		ExchangeData(	ADR(Parameters.Regulation.ExtractAir.ControlMode), 
						ADR(ADS_Standard.Tags.Settings.ExtractFanControlMode), 
						SIZEOF(Parameters.Regulation.ExtractAir.ControlMode), 
						ADR(SavedParameters.Regulation.Temperature.TemperatureControlSource), 
						ADR(SavedInterface.ExtractFanControlMode), 
						'INT', ('Parameters.Regulation.ExtractAir.ControlMode'), ('ExtractFanControlMode'));	
		
		ExchangeData_LREAL_REAL(	ADR(Parameters.Regulation.ExtractAir.Control.SP), 
						ADR(ADS_Standard.Tags.Settings.ExtractFan_SP), 
						ADR(SavedParameters.Regulation.ExtractAir.Control.SP), 
						ADR(SavedInterface.ExtractFan_SP), 
						('Parameters.Regulation.ExtractAir.Control.SP'), ('ExtractFan_SP'));	
		
		ExchangeData_LREAL_REAL(	ADR(Parameters.Regulation.ExtractAir.Control.SP_HighSpeed), 
						ADR(ADS_Standard.Tags.Settings.ExtractFanHighSpeed_SP), 
						ADR(SavedParameters.Regulation.ExtractAir.Control.SP_HighSpeed), 
						ADR(SavedInterface.ExtractFanHighSpeed_SP), 
						('Parameters.Regulation.ExtractAir.Control.SP_HighSpeed'), ('ExtractFanHighSpeed_SP'));	
		
		ExchangeData_LREAL_REAL(	ADR(Parameters.Regulation.ExtractAir.Control.P), 
						ADR(ADS_Standard.Tags.Settings.ExtractFanControl_P), 
						ADR(SavedParameters.Regulation.ExtractAir.Control.P), 
						ADR(SavedInterface.ExtractFanControl_P), 
						('Parameters.Regulation.ExtractAir.Control.P'), ('ExtractFanControl_P'));	
		
		ExchangeData(	ADR(Parameters.Regulation.ExtractAir.Control.I), 
						ADR(ADS_Standard.Tags.Settings.ExtractFanControl_I), 
						SIZEOF(Parameters.Regulation.ExtractAir.Control.I),
						ADR(SavedParameters.Regulation.ExtractAir.Control.I), 
						ADR(SavedInterface.ExtractFanControl_I), 
						'TIME', ('Parameters.Regulation.ExtractAir.Control.I'), ('ExtractFanControl_I'));	
		
		ExchangeData(	ADR(Parameters.Regulation.ExtractAir.SetPointAdjustment.Curve), 
						ADR(ADS_Standard.Tags.Settings.F_GQ1_CURVE), 
						SIZEOF(Parameters.Regulation.ExtractAir.SetPointAdjustment.Curve), 
						ADR(SavedParameters.Regulation.ExtractAir.SetPointAdjustment.Curve), 
						ADR(SavedInterface.F_GQ1_CURVE), 
						'SetPointOffsetCurve', ('Parameters.Regulation.ExtractAir.SetPointAdjustment.Curve'), ('F_GQ1_CURVE'));	
		
		// TBD ExchangeData !!!!!!!!!!!!!!!!!!!!!!!!!!!!!!!!!!!!
		
		ExchangeData(	ADR(Parameters.Alarm.Delay.B.RegulationDeviation), 
						ADR(ADS_Standard.Tags.Settings.T_BT1_AD), 
						SIZEOF(Parameters.Alarm.Delay.B.RegulationDeviation), 
						ADR(SavedParameters.Alarm.Delay.B.RegulationDeviation), 
						ADR(SavedInterface.T_BT1_AD), 
						'TIME', ('Parameters.Alarm.Delay.B.RegulationDeviation'), ('T_BT1_AD'));	
		// ADS_Standard.Tags.Settings.T_BT1_AD := Parameters.Alarm.Delay.B.RegulationDeviation;
		
		ExchangeData(	ADR(Parameters.Alarm.Limits.B.RegulationDeviation), 
						ADR(ADS_Standard.Tags.Settings.T_BT1_ADL), 
						SIZEOF(Parameters.Alarm.Limits.B.RegulationDeviation), 
						ADR(SavedParameters.Alarm.Limits.B.RegulationDeviation), 
						ADR(SavedInterface.T_BT1_ADL), 
						'REAL', ('Parameters.Alarm.Limits.B.RegulationDeviation'), ('T_BT1_ADL'));	
		// ADS_Standard.Tags.Settings.T_BT1_ALL := Parameters.Alarm.Limits.B.RegulationDeviation;
		
		ExchangeData(	ADR(Parameters.Alarm.Delay.B.SupplyFan), 
						ADR(ADS_Standard.Tags.Settings.T_GQ1_AD), 
						SIZEOF(Parameters.Alarm.Delay.B.SupplyFan), 
						ADR(SavedParameters.Alarm.Delay.B.SupplyFan), 
						ADR(SavedInterface.T_GQ1_AD), 
						'TIME', ('Parameters.Alarm.Delay.B.SupplyFan'), ('T_GQ1_AD'));	
		// ADS_Standard.Tags.Settings.T_GQ1_AD := Parameters.Alarm.Delay.B.SupplyFan;
		
		ExchangeData(	ADR(Parameters.Alarm.Delay.B.ExtractFan), 
						ADR(ADS_Standard.Tags.Settings.F_GQ1_AD), 
						SIZEOF(Parameters.Alarm.Delay.B.ExtractFan), 
						ADR(SavedParameters.Alarm.Delay.B.ExtractFan), 
						ADR(SavedInterface.F_GQ1_AD), 
						'TIME', ('Parameters.Alarm.Delay.B.ExtractFan'), ('F_GQ1_AD'));	
		// ADS_Standard.Tags.Settings.F_GQ1_AD := Parameters.Alarm.Delay.B.ExtractFan;
		
		ExchangeData(	ADR(Parameters.Alarm.Delay.B.SupplyFilter), 
						ADR(ADS_Standard.Tags.Settings.T_BP2_AD), 
						SIZEOF(Parameters.Alarm.Delay.B.SupplyFilter), 
						ADR(SavedParameters.Alarm.Delay.B.SupplyFilter), 
						ADR(SavedInterface.T_BP2_AD), 
						'TIME', ('Parameters.Alarm.Delay.B.SupplyFilter'), ('T_BP2_AD'));	
		// ADS_Standard.Tags.Settings.T_BP2_AD := Parameters.Alarm.Delay.B.SupplyFilter;
		
		ExchangeData(	ADR(Parameters.Alarm.Limits.B.SupplyFilter), 
						ADR(ADS_Standard.Tags.Settings.T_BP2_AHL), 
						SIZEOF(Parameters.Alarm.Limits.B.SupplyFilter), 
						ADR(SavedParameters.Alarm.Limits.B.SupplyFilter), 
						ADR(SavedInterface.T_BP2_AHL), 
						'REAL', ('Parameters.Alarm.Limits.B.SupplyFilter'), ('T_BP2_AHL'));	
		// ADS_Standard.Tags.Settings.T_BP2_HLL := Parameters.Alarm.Limits.B.SupplyFilter;
		
		ExchangeData(	ADR(Parameters.Alarm.Delay.B.ExtractFilter), 
						ADR(ADS_Standard.Tags.Settings.F_BP2_AD), 
						SIZEOF(Parameters.Alarm.Delay.B.ExtractFilter), 
						ADR(SavedParameters.Alarm.Delay.B.ExtractFilter), 
						ADR(SavedInterface.F_BP2_AD), 
						'TIME', ('Parameters.Alarm.Delay.B.ExtractFilter'), ('F_BP2_AD'));	
		// ADS_Standard.Tags.Settings.F_BP2_AD := Parameters.Alarm.Delay.B.ExtractFilter;
		
		ExchangeData(	ADR(Parameters.Alarm.Limits.B.ExtractFilter), 
						ADR(ADS_Standard.Tags.Settings.F_BP2_AHL), 
						SIZEOF(Parameters.Alarm.Limits.B.ExtractFilter), 
						ADR(SavedParameters.Alarm.Limits.B.ExtractFilter), 
						ADR(SavedInterface.F_BP2_AHL), 
						'REAL', ('Parameters.Alarm.Limits.B.ExtractFilter'), ('F_BP2_AHL'));	
		// ADS_Standard.Tags.Settings.F_BP2_HLL := Parameters.Alarm.Limits.B.ExtractFilter;
		
		ExchangeData(	ADR(Parameters.System.Exercise.FireBypassDamper.Interval), 
						ADR(ADS_Standard.Tags.Settings.F_QM2_SP1), 
						SIZEOF(Parameters.System.Exercise.FireBypassDamper.Interval), 
						ADR(SavedParameters.System.Exercise.FireBypassDamper.Interval), 
						ADR(SavedInterface.F_QM2_SP1), 
						'INT', ('Parameters.System.Exercise.FireBypassDamper.Interval'), ('F_QM2_SP1'));	
		// ADS_Standard.Tags.Settings.F_QM2_XI := Parameters.System.Exercise.FireBypassDamper.Interval;
		
		ExchangeData(	ADR(Parameters.System.Exercise.FireBypassDamper.Hour), 
						ADR(ADS_Standard.Tags.Settings.F_QM2_SP2), 
						SIZEOF(Parameters.System.Exercise.FireBypassDamper.Hour), 
						ADR(SavedParameters.System.Exercise.FireBypassDamper.Hour), 
						ADR(SavedInterface.F_QM2_SP2), 
						'INT', ('Parameters.System.Exercise.FireBypassDamper.Hour'), ('F_QM2_SP2'));
	
		ExchangeData(	ADR(Parameters.System.Exercise.FireBypassDamper.Minute), 
						ADR(ADS_Standard.Tags.Settings.F_QM2_SP3), 
						SIZEOF(Parameters.System.Exercise.FireBypassDamper.Minute), 
						ADR(SavedParameters.System.Exercise.FireBypassDamper.Minute), 
						ADR(SavedInterface.F_QM2_SP3), 
						'INT', ('Parameters.System.Exercise.FireBypassDamper.Minute'), ('F_QM2_SP3'));
						
		ExchangeData(	ADR(ParametersSC.NetLink.Exercise.Interval), 
						ADR(ADS_Standard.Tags.Settings.EXT_QM_SP1), 
						SIZEOF(ParametersSC.NetLink.Exercise.Interval), 
						ADR(SavedParametersSC.NetLink.Exercise.Interval), 
						ADR(SavedInterface.EXT_QM_SP1), 
						'INT', ('ParametersSC.NetLink.Exercise.Interval'), ('EXT_QM_SP1'));	
		// ADS_Standard.Tags.Settings.EXT_QM_XI := ParametersSC.NetLink.Exercise.Interval;
		
		ExchangeData(	ADR(ParametersSC.NetLink.Exercise.Hour), 
						ADR(ADS_Standard.Tags.Settings.EXT_QM_SP2), 
						SIZEOF(ParametersSC.NetLink.Exercise.Hour), 
						ADR(SavedParametersSC.NetLink.Exercise.Hour), 
						ADR(SavedInterface.EXT_QM_SP2), 
						'INT', ('ParametersSC.NetLink.Exercise.Hour'), ('EXT_QM_SP2'));
		ExchangeData(	ADR(ParametersSC.NetLink.Exercise.Minute), 
						ADR(ADS_Standard.Tags.Settings.EXT_QM_SP3), 
						SIZEOF(ParametersSC.NetLink.Exercise.Minute), 
						ADR(SavedParametersSC.NetLink.Exercise.Minute), 
						ADR(SavedInterface.EXT_QM_SP3), 
						'INT', ('ParametersSC.NetLink.Exercise.Minute'), ('EXT_QM_SP3'));	
	
		ExchangeData(	ADR(Parameters.Alarm.Delay.B.SupplyAirDeviation), 
						ADR(ADS_Standard.Tags.Settings.T_BP1_AD), 
						SIZEOF(Parameters.Alarm.Delay.B.SupplyAirDeviation), 
						ADR(SavedParameters.Alarm.Delay.B.SupplyAirDeviation), 
						ADR(SavedInterface.T_BP1_AD), 
						'TIME', ('Parameters.Alarm.Delay.B.SupplyAirDeviation'), ('T_BP1_AD'));	
		
		ExchangeData(	ADR(Parameters.Alarm.Limits.B.SupplyAirPressureDeviation), 
						ADR(ADS_Standard.Tags.Settings.T_BP1_ADL), 
						SIZEOF(Parameters.Alarm.Limits.B.SupplyAirPressureDeviation), 
						ADR(SavedParameters.Alarm.Limits.B.SupplyAirPressureDeviation), 
						ADR(SavedInterface.T_BP1_ADL), 
						'REAL', ('Parameters.Alarm.Limits.B.SupplyAirPressureDeviation'), ('T_BP1_ADL'));	
		
		ExchangeData(	ADR(Parameters.Alarm.Delay.B.ExtractAirDeviation), 
						ADR(ADS_Standard.Tags.Settings.F_BP1_AD), 
						SIZEOF(Parameters.Alarm.Delay.B.ExtractAirDeviation), 
						ADR(SavedParameters.Alarm.Delay.B.ExtractAirDeviation), 
						ADR(SavedInterface.F_BP1_AD), 
						'TIME', ('Parameters.Alarm.Delay.B.ExtractAirDeviation'), ('F_BP1_AD'));	
		
		ExchangeData(	ADR(Parameters.Alarm.Limits.B.ExtractAirPressureDeviation), 
						ADR(ADS_Standard.Tags.Settings.F_BP1_ADL), 
						SIZEOF(Parameters.Alarm.Limits.B.ExtractAirPressureDeviation), 
						ADR(SavedParameters.Alarm.Limits.B.ExtractAirPressureDeviation), 
						ADR(SavedInterface.F_BP1_ADL), 
						'REAL', ('Parameters.Alarm.Limits.B.ExtractAirPressureDeviation'), ('F_BP1_ADL'));	

		ExchangeData(	ADR(Parameters.Alarm.Limits.A.Freeze), 
						ADR(ADS_Standard.Tags.Settings.FREEZE_ALL), 
						SIZEOF(Parameters.Alarm.Limits.A.Freeze), 
						ADR(SavedParameters.Alarm.Limits.A.Freeze), 
						ADR(SavedInterface.FREEZE_ALL), 
						'REAL', ('Parameters.Alarm.Limits.A.Freeze'), ('FREEZE_ALL'));	

		Parameters.IO.AOutOverride.T_GQ1_Override := ADS_Standard.Tags.Settings.T_GQ1_M;
		Parameters.IO.AOutOverride.T_GQ1_OverrideValue := ADS_Standard.Tags.Settings.T_GQ1_OPM;			
		Parameters.IO.AOutOverride.F_GQ1_Override := ADS_Standard.Tags.Settings.F_GQ1_M;
		Parameters.IO.AOutOverride.F_GQ1_OverrideValue := ADS_Standard.Tags.Settings.F_GQ1_OPM;			
		Parameters.IO.AOutOverride.H_QN1_Override := ADS_Standard.Tags.Settings.H_QN1_M;
		Parameters.IO.AOutOverride.H_QN1_OverrideValue := ADS_Standard.Tags.Settings.H_QN1_OPM;			
		Parameters.IO.AOutOverride.F_QN1_Override := ADS_Standard.Tags.Settings.TX1_M;
		Parameters.IO.AOutOverride.F_QN1_OverrideValue := ADS_Standard.Tags.Settings.TX1_OPM;			
		Parameters.IO.AOutOverride.C_QN1_Override := ADS_Standard.Tags.Settings.C_QN1_M;
		Parameters.IO.AOutOverride.C_QN1_OverrideValue := ADS_Standard.Tags.Settings.C_QN1_OPM;		

		Parameters.IO.DOutOverride.H_GP1_Override := ADS_Standard.Tags.Settings.H_GP1_M;	
		Parameters.IO.DOutOverride.C_GP1_Override := ADS_Standard.Tags.Settings.C_GP1_M;
		Parameters.IO.DOutOverride.F_QM1_Override := ADS_Standard.Tags.Settings.F_QM1_M;
		Parameters.IO.DOutOverride.T_QM1_1_Override := ADS_Standard.Tags.Settings.T_QM1_1_M;
		Parameters.IO.DOutOverride.T_QM1_2_Override := ADS_Standard.Tags.Settings.T_QM1_2_M;
		Parameters.IO.DOutOverride.T_QM1_3_Override := ADS_Standard.Tags.Settings.T_QM1_3_M;
		Parameters.IO.DOutOverride.T_QM1_4_Override := ADS_Standard.Tags.Settings.T_QM1_4_M;
		Parameters.IO.DOutOverride.T_QM1_5_Override := ADS_Standard.Tags.Settings.T_QM1_5_M;
		Parameters.IO.DOutOverride.T_QM1_6_Override := ADS_Standard.Tags.Settings.T_QM1_6_M;
		Parameters.IO.DOutOverride.F_QM2_Override := ADS_Standard.Tags.Settings.F_QM2_M;
		Parameters.IO.DOutOverride.T_QM2_Override := ADS_Standard.Tags.Settings.T_QM2_M;
		
		Parameters.IO.DOutOverride.H_GP1_OverrideValue := ADS_Standard.Tags.Settings.H_GP1_MCMD;	
		Parameters.IO.DOutOverride.C_GP1_OverrideValue := ADS_Standard.Tags.Settings.C_GP1_MCMD;
		Parameters.IO.DOutOverride.F_QM1_OverrideValue := ADS_Standard.Tags.Settings.F_QM1_MCMD;
		Parameters.IO.DOutOverride.T_QM1_1_OverrideValue := ADS_Standard.Tags.Settings.T_QM1_1_MCMD;
		Parameters.IO.DOutOverride.T_QM1_2_OverrideValue := ADS_Standard.Tags.Settings.T_QM1_2_MCMD;
		Parameters.IO.DOutOverride.T_QM1_3_OverrideValue := ADS_Standard.Tags.Settings.T_QM1_3_MCMD;
		Parameters.IO.DOutOverride.T_QM1_4_OverrideValue := ADS_Standard.Tags.Settings.T_QM1_4_MCMD;
		Parameters.IO.DOutOverride.T_QM1_5_OverrideValue := ADS_Standard.Tags.Settings.T_QM1_5_MCMD;
		Parameters.IO.DOutOverride.T_QM1_6_OverrideValue := ADS_Standard.Tags.Settings.T_QM1_6_MCMD;
		Parameters.IO.DOutOverride.F_QM2_OverrideValue := ADS_Standard.Tags.Settings.F_QM2_MCMD;
		Parameters.IO.DOutOverride.T_QM2_OverrideValue := ADS_Standard.Tags.Settings.T_QM2_MCMD;
	END_IF
	
	// Status transfers
	ADS_Standard.Tags.Status.ENO := Parameters.System.Operation.ENO;
	ADS_Standard.Tags.Status.Auto := Parameters.IO.DIn.Auto;
	ADS_Standard.Tags.Status.Hand := Parameters.IO.DIn.Hand;
	ADS_Standard.Tags.Status.TX1_EFF_LAL := Parameters.Alarm.Active.B.HeatExchangerEfficiency;
	ADS_Standard.Tags.Status.SFP_PV := TO_REAL(Parameters.Regulation.SystemSpecificFanPower);
	ADS_Standard.Tags.Status.TC_V := Parameters.System.Operation.TimeChannels.Q;
	ADS_Standard.Tags.Status.F_BR1_AL := Parameters.Alarm.Active.A.FireExtract; // GM_XXL.DI.FireExtractAlarm;
	ADS_Standard.Tags.Status.F_BRT2_AL := Parameters.Alarm.Active.A.FireExtractTemperature;
	ADS_Standard.Tags.Status.F_BRT3_AL := Parameters.Alarm.Active.A.FireExtractPressure;
	ADS_Standard.Tags.Status.T_BR1_AL := Parameters.Alarm.Active.A.FireSupply;
	ADS_Standard.Tags.Status.F_BR1_FAULT := Parameters.Alarm.Active.B.SmokeDetectorServiceExtract;
	ADS_Standard.Tags.Status.T_BR1_FAULT := Parameters.Alarm.Active.B.SmokeDetectorServiceSupply;
	
	ADS_Standard.Tags.Status.F_BP1_AL := Parameters.Alarm.Active.B.ExtractAirDeviation;
	ADS_Standard.Tags.Status.T_BP1_AL := Parameters.Alarm.Active.B.SupplyAirDeviation;
	ADS_Standard.Tags.Status.T_BT1_AL := Parameters.Alarm.Active.B.RegulationDeviation;
	
	ADS_Standard.Tags.Status.H_BT1_LAL := Parameters.Alarm.Active.A.Freeze;
	
	ADS_Standard.Tags.Status.BT1_FAULT := Parameters.IO.AIn.BT1_Error;
	ADS_Standard.Tags.Status.BT2_FAULT := Parameters.IO.AIn.BT2_Error;
	ADS_Standard.Tags.Status.F_BF1_FAULT := Parameters.IO.AIn.F_BF1_Error;
	ADS_Standard.Tags.Status.F_BP1_FAULT := Parameters.IO.AIn.F_BP1_Error;
	ADS_Standard.Tags.Status.F_BP2_FAULT := Parameters.IO.AIn.F_BP2_Error;
	ADS_Standard.Tags.Status.F_BP3_FAULT := Parameters.IO.AIn.F_BP3_Error;
	ADS_Standard.Tags.Status.F_BT1_FAULT := Parameters.IO.AIn.F_BT1_Error;
	ADS_Standard.Tags.Status.F_BT2_FAULT := Parameters.IO.AIn.F_BT2_Error;
	ADS_Standard.Tags.Status.H_BT1_FAULT := Parameters.IO.AIn.H_BT1_Error;
	ADS_Standard.Tags.Status.T_BF1_FAULT := Parameters.IO.AIn.T_BF1_Error;
	ADS_Standard.Tags.Status.T_BP1_FAULT := Parameters.IO.AIn.T_BP1_Error;
	ADS_Standard.Tags.Status.T_BP2_FAULT := Parameters.IO.AIn.T_BP2_Error;
	ADS_Standard.Tags.Status.T_BT1_FAULT := Parameters.IO.AIn.T_BT1_Error;
	ADS_Standard.Tags.Status.T_BT2_FAULT := Parameters.IO.AIn.T_BT2_Error;
	ADS_Standard.Tags.Status.T_BT3_FAULT := Parameters.IO.AIn.T_BT3_Error;
	
	ADS_Standard.Tags.Status.Fuse_AL := Parameters.Alarm.Active.A.Fuse;
	ADS_Standard.Tags.Status.T_GQ1_AL := Parameters.Alarm.Active.B.SupplyFan;
	ADS_Standard.Tags.Status.F_GQ1_AL := Parameters.Alarm.Active.B.ExtractFan;
	ADS_Standard.Tags.Status.Fire_AL := Parameters.Alarm.Active.A.FireExtract OR
											Parameters.Alarm.Active.A.FireExtractExternal OR
											Parameters.Alarm.Active.A.FireExtractPressure OR
											Parameters.Alarm.Active.A.FireExtractTemperature OR
											Parameters.Alarm.Active.A.FireLocal OR
											Parameters.Alarm.Active.A.FireSupply;
	ADS_Standard.Tags.Status.H_GP1_V := Parameters.IO.DIn.H_GP1_Running;
	ADS_Standard.Tags.Status.H_GP1_AL := Parameters.Alarm.Active.B.Pump1;
	ADS_Standard.Tags.Status.C_GP1_V := Parameters.IO.DIn.C_GP1_Running;
	ADS_Standard.Tags.Status.C_GP1_AL := Parameters.Alarm.Active.B.Pump2;
	ADS_Standard.Tags.Status.T_BP2_HAL := Parameters.Alarm.Active.B.SupplyFilter;
	ADS_Standard.Tags.Status.F_BP2_HAL := Parameters.Alarm.Active.B.ExtractFilter;
	
	ADS_Standard.Tags.Status.H_GP1_CMD := Main.GreenMasterDO.H_GP1;
	ADS_Standard.Tags.Status.C_GP1_CMD := Main.GreenMasterDO.C_GP1;
	ADS_Standard.Tags.Status.F_QM1_CMD := Main.GreenMasterDO.F_QM1;
	ADS_Standard.Tags.Status.T_QM2_CMD := Main.GreenMasterDO.T_QM2;
	(*!!!!! BORT !!!! *)ADS_Standard.Tags.Status.T_QM3_CMD := Main.GreenMasterDO.T_QM2;
		
	ADS_Standard.Tags.Status.F_QM2_CMD := Main.GreenMasterDO.F_QM2;
	ADS_Standard.Tags.Status.F_QM2_V0 := Parameters.IO.DIn.F_QM2_Closed;
	ADS_Standard.Tags.Status.F_QM2_V1 := Parameters.IO.DIn.F_QM2_Open;
	
	ADS_Standard.Tags.Status.T_QM1_1_CMD := Main.GreenMasterDO.T_QM1_1;
	ADS_Standard.Tags.Status.T_QM1_2_CMD := Main.GreenMasterDO.T_QM1_2;
	ADS_Standard.Tags.Status.T_QM1_3_CMD := Main.GreenMasterDO.T_QM1_3;
	ADS_Standard.Tags.Status.T_QM1_4_CMD := Main.GreenMasterDO.T_QM1_4;
	ADS_Standard.Tags.Status.T_QM1_5_CMD := Main.GreenMasterDO.T_QM1_5;
	ADS_Standard.Tags.Status.T_QM1_6_CMD := Main.GreenMasterDO.T_QM1_6;

	ADS_Standard.Tags.Status.T_QM1_CMD := Main.GreenMasterDO.T_QM2;

	ADS_Standard.Tags.Status.Temperature_CSP := LREAL_TO_REAL(Parameters.Regulation.Temperature.Control.CSP);
	ADS_Standard.Tags.Status.T_BP1_CSP := LREAL_TO_REAL(Parameters.Regulation.SupplyAir.Control.CSP);
	ADS_Standard.Tags.Status.F_BP1_CSP := LREAL_TO_REAL(Parameters.Regulation.ExtractAir.Control.CSP);
	ADS_Standard.Tags.Status.F_BT1_PV := LREAL_TO_REAL(Parameters.IO.AIn.F_BT1);
	ADS_Standard.Tags.Status.T_BT2_PV := LREAL_TO_REAL(Parameters.IO.AIn.T_BT2);
	ADS_Standard.Tags.Status.T_BT3_PV := LREAL_TO_REAL(Parameters.IO.AIn.T_BT3);
	ADS_Standard.Tags.Status.H_BT1_PV := LREAL_TO_REAL(Parameters.IO.AIn.H_BT1);
	ADS_Standard.Tags.Status.T_BT1_PV := LREAL_TO_REAL(Parameters.IO.AIn.T_BT1);
	ADS_Standard.Tags.Status.F_BT2_PV := LREAL_TO_REAL(Parameters.IO.AIn.F_BT2);
	
	IF NOT Parameters.IO.AIn.T_BF1_Error THEN
		ADS_Standard.Tags.Status.T_BF1_PV := LREAL_TO_REAL(Parameters.IO.AIn.T_BF1);
	ELSE	
		ADS_Standard.Tags.Status.T_BF1_PV := 0;
	END_IF
	IF NOT Parameters.IO.AIn.F_BF1_Error THEN
		ADS_Standard.Tags.Status.F_BF1_PV := LREAL_TO_REAL(Parameters.IO.AIn.F_BF1);
	ELSE	
		ADS_Standard.Tags.Status.F_BF1_PV := 0;
	END_IF
	ADS_Standard.Tags.Status.T_BP1_PV := LREAL_TO_REAL(Parameters.IO.AIn.T_BP1);
	ADS_Standard.Tags.Status.F_BP1_PV := LREAL_TO_REAL(Parameters.IO.AIn.F_BP1);
	ADS_Standard.Tags.Status.T_BP2_PV := LREAL_TO_REAL(Parameters.IO.AIn.T_BP2);
	ADS_Standard.Tags.Status.F_BP2_PV := LREAL_TO_REAL(Parameters.IO.AIn.F_BP2);
	ADS_Standard.Tags.Status.F_BP3_PV := LREAL_TO_REAL(Parameters.IO.AIn.F_BP3);
	
	ADS_Standard.Tags.Status.TX1_OP := TO_REAL(Main.GreenMasterAO.F_QN1); //LREAL_TO_REAL(Parameters.IO.AOut.F_QN1);
	ADS_Standard.Tags.Status.H_QN1_OP := LREAL_TO_REAL(Main.GreenMasterAO.H_QN1);
	ADS_Standard.Tags.Status.C_QN1_OP := LREAL_TO_REAL(Main.GreenMasterAO.C_QN1);
	ADS_Standard.Tags.Status.T_GQ1_OP := LREAL_TO_REAL(Main.GreenMasterAO.T_GQ1);
	ADS_Standard.Tags.Status.F_GQ1_OP := LREAL_TO_REAL(Main.GreenMasterAO.F_GQ1);
	ADS_Standard.Tags.Status.T_GQ1_V := Parameters.IO.AOut.T_GQ1 > 0.02;
	ADS_Standard.Tags.Status.F_GQ1_V := Parameters.IO.AOut.F_GQ1 > 0.02;
	
	ADS_Standard.Tags.Status.TX1_EFF_PV := LREAL_TO_REAL(Parameters.Regulation.Temperature.Efficiency);
	ADS_Standard.Tags.Status.TX1_EFF_LAL := Parameters.Alarm.Active.B.HeatExchangerEfficiency;
	ADS_Standard.Tags.Status.PLC_VERSION_PV := GlobalSettings.PlcVersion;
	ADS_Standard.Tags.Status.TIMEANDDATE_PV := Parameters.System.SystemTime;
	ADS_Standard.Tags.Status.NightCooling_V := Parameters.Regulation.NightCooling;
	ADS_Standard.Tags.Status.TX1_AL := Parameters.Alarm.Active.B.Tx1Fail;
	
	PreEN := TRUE;
	
	ModbusSettings();
	ModbusStatus();
ELSE
	IF PreEN THEN
		Globals.IO.DOut.DO16 := FALSE;
	END_IF
	PreEN := FALSE;
END_IF

METHOD ExchangeData : BOOL
VAR_INPUT
	PData1: POINTER TO BYTE;
	PData2: POINTER TO BYTE;
	Size: UDINT;
	PSavedData1: POINTER TO BYTE;
	PSavedData2: POINTER TO BYTE;
	VarType: STRING;
	{attribute 'TcEncoding':='UTF-8'}
	LogText1: STRING := '';
	{attribute 'TcEncoding':='UTF-8'}
	LogText2: STRING := '';
END_VAR
VAR
END_VAR
IF MemCmp(PData1, PSavedData1, Size) <> 0 THEN
	MemCpy(PData2, PData1, Size);
	MemCpy(PSavedData2, PData1, Size);
	MemCpy(PSavedData1, PData1, Size);
	IF LogText1 <> '' THEN
		Main.EventLog.LogEventJSON(EventTypes.Information, concat('Local change ', concat(concat(LogText1, ' => '), LogText2)), VarType, Size, PData1);	
	END_IF
END_IF
IF MemCmp(PData2, PSavedData2, Size) <> 0 THEN
	MemCpy(PData1, PData2, Size);
	MemCpy(PSavedData1, PData2, Size);
	MemCpy(PSavedData2, PData2, Size);
	IF LogText2 <> '' THEN
		Main.EventLog.LogEventJSON(EventTypes.Information, concat('ADS change ', concat(concat(LogText2, ' => '), LogText1)), VarType, Size, PData2);	
	END_IF
END_IF
END_METHOD

METHOD ExchangeData_LREAL_REAL : BOOL
VAR_INPUT
	PData1: POINTER TO LREAL;
	PData2: POINTER TO REAL;
	PSavedData1: POINTER TO LREAL;
	PSavedData2: POINTER TO REAL;
	{attribute 'TcEncoding':='UTF-8'}
	LogText1: STRING := '';
	{attribute 'TcEncoding':='UTF-8'}
	LogText2: STRING := '';
END_VAR
VAR
END_VAR
IF PData1^ <> PSavedData1^ THEN
	PData2^ := TO_REAL(PData1^);
	PSavedData2^ := TO_REAL(PData1^);
	PSavedData1^ := PData1^;
	IF LogText1 <> '' THEN
		Main.EventLog.LogEventJSON(EventTypes.Information, concat('Local change ', concat(concat(LogText1, ' => '), LogText2)), 'LREAL', SIZEOF(LREAL), PData1);	
	END_IF
END_IF
IF PData2^ <> PSavedData2^ THEN
	PData1^ := TO_LREAL(PData2^);
	PSavedData1^ := TO_LREAL(PData2^);
	PSavedData2^ := PData2^;
	IF LogText2 <> '' THEN
		Main.EventLog.LogEventJSON(EventTypes.Information, concat('ADS change ', concat(concat(LogText2, ' => '), LogText1)), 'REAL', SIZEOF(REAL), PData2);	
	END_IF
END_IF
END_METHOD

METHOD ModbusSettings : BOOL
VAR_INPUT
END_VAR
GVL.mb_Output_Registers[0] := BOOL_TO_WORD(ADS_Standard.Tags.Status.TC_V);
END_METHOD

ACTION ModbusStatus:
GVL.mb_Input_Registers[0] := REAL_TO_WORD_SAFE(ADS_Standard.Tags.Status.TEMPERATURE_CSP);

GVL.mb_Input_Registers[100] := REAL_TO_WORD_SAFE(ADS_Standard.Tags.Status.BT1_PV * 10);
GVL.mb_Input_Registers[101] := REAL_TO_WORD_SAFE(ADS_Standard.Tags.Status.T_BT2_PV * 10);
GVL.mb_Input_Registers[102] := REAL_TO_WORD_SAFE(ADS_Standard.Tags.Status.T_BT3_PV * 10);
GVL.mb_Input_Registers[103] := REAL_TO_WORD_SAFE(ADS_Standard.Tags.Status.H_BT1_PV * 10);
GVL.mb_Input_Registers[104] := REAL_TO_WORD_SAFE(ADS_Standard.Tags.Status.T_BT1_PV * 10);
GVL.mb_Input_Registers[105] := REAL_TO_WORD_SAFE(ADS_Standard.Tags.Status.F_BT1_PV * 10);
GVL.mb_Input_Registers[106] := REAL_TO_WORD_SAFE(ADS_Standard.Tags.Status.F_BT2_PV * 10);
GVL.mb_Input_Registers[107] := REAL_TO_WORD_SAFE(ADS_Standard.Tags.Status.BT2_PV * 10);

GVL.mb_Input_Registers[200] := REAL_TO_WORD_SAFE(ADS_Standard.Tags.Status.T_BP1_CSP);
GVL.mb_Input_Registers[201] := REAL_TO_WORD_SAFE(ADS_Standard.Tags.Status.F_BP1_CSP);

GVL.mb_Input_Registers[300] := REAL_TO_WORD_SAFE(ADS_Standard.Tags.Status.T_BP1_PV);
GVL.mb_Input_Registers[301] := REAL_TO_WORD_SAFE(ADS_Standard.Tags.Status.F_BP1_PV);

GVL.mb_Input_Registers[500] := REAL_TO_WORD_SAFE(ADS_Standard.Tags.Status.T_BF1_PV);
GVL.mb_Input_Registers[501] := REAL_TO_WORD_SAFE(ADS_Standard.Tags.Status.F_BF1_PV);

GVL.mb_Input_Registers[600] := REAL_TO_WORD_SAFE(ADS_Standard.Tags.Status.TX1_EFF_PV * 100);
GVL.mb_Input_Registers[601] := REAL_TO_WORD_SAFE(ADS_Standard.Tags.Status.SFP_PV * 1000);

GVL.mb_Input_Registers[700] := REAL_TO_WORD_SAFE(ADS_Standard.Tags.Status.T_GQ1_OP * 100);
GVL.mb_Input_Registers[701] := REAL_TO_WORD_SAFE(ADS_Standard.Tags.Status.F_GQ1_OP * 100);
GVL.mb_Input_Registers[702] := REAL_TO_WORD_SAFE(ADS_Standard.Tags.Status.TX1_OP * 100);
GVL.mb_Input_Registers[703] := REAL_TO_WORD_SAFE(ADS_Standard.Tags.Status.H_QN1_OP * 100);
GVL.mb_Input_Registers[704] := REAL_TO_WORD_SAFE(ADS_Standard.Tags.Status.C_QN1_OP * 100);

GVL.mb_Input_Registers[800] := BOOL_TO_WORD(ADS_Standard.Tags.Status.T_GQ1_OP > 0);
GVL.mb_Input_Registers[801] := BOOL_TO_WORD(ADS_Standard.Tags.Status.F_GQ1_OP > 0);
GVL.mb_Input_Registers[802] := BOOL_TO_WORD(ADS_Standard.Tags.Status.H_GP1_CMD);
GVL.mb_Input_Registers[803] := BOOL_TO_WORD(ADS_Standard.Tags.Status.C_GP1_CMD);

GVL.mb_Input_Registers[900] := BOOL_TO_WORD(ADS_Standard.Tags.Status.F_BR1_AL);
GVL.mb_Input_Registers[901] := BOOL_TO_WORD(ADS_Standard.Tags.Status.T_BR1_AL);
GVL.mb_Input_Registers[902] := BOOL_TO_WORD(ADS_Standard.Tags.Status.FIRE_AL);
GVL.mb_Input_Registers[903] := BOOL_TO_WORD(ADS_Standard.Tags.Status.F_BRT2_AL);
GVL.mb_Input_Registers[904] := BOOL_TO_WORD(ADS_Standard.Tags.Status.F_BRT3_AL);
GVL.mb_Input_Registers[905] := BOOL_TO_WORD(ADS_Standard.Tags.Status.FUSE_AL);
GVL.mb_Input_Registers[906] := BOOL_TO_WORD(ADS_Standard.Tags.Status.T_GQ1_AL);
GVL.mb_Input_Registers[907] := BOOL_TO_WORD(ADS_Standard.Tags.Status.T_GQ_AL1);
GVL.mb_Input_Registers[908] := BOOL_TO_WORD(ADS_Standard.Tags.Status.T_GQ_AL2);
GVL.mb_Input_Registers[909] := BOOL_TO_WORD(ADS_Standard.Tags.Status.F_GQ1_AL);
GVL.mb_Input_Registers[910] := BOOL_TO_WORD(ADS_Standard.Tags.Status.F_GQ_AL1);
GVL.mb_Input_Registers[911] := BOOL_TO_WORD(ADS_Standard.Tags.Status.F_GQ_AL2);
GVL.mb_Input_Registers[912] := BOOL_TO_WORD(ADS_Standard.Tags.Status.H_GP1_AL);
GVL.mb_Input_Registers[913] := BOOL_TO_WORD(ADS_Standard.Tags.Status.C_GP1_AL);
GVL.mb_Input_Registers[914] := BOOL_TO_WORD(ADS_Standard.Tags.Status.QM_AL);
GVL.mb_Input_Registers[915] := BOOL_TO_WORD(ADS_Standard.Tags.Status.TX1_EFF_LAL);
GVL.mb_Input_Registers[916] := BOOL_TO_WORD(ADS_Standard.Tags.Status.H_BT1_LAL);
GVL.mb_Input_Registers[917] := BOOL_TO_WORD(ADS_Standard.Tags.Status.T_BP2_HAL);
GVL.mb_Input_Registers[918] := BOOL_TO_WORD(ADS_Standard.Tags.Status.F_BP2_HAL);
GVL.mb_Input_Registers[919] := BOOL_TO_WORD(ADS_Standard.Tags.Status.F_BP3_AL);
GVL.mb_Input_Registers[920] := BOOL_TO_WORD(ADS_Standard.Tags.Status.T_BT3_FAULT);
GVL.mb_Input_Registers[921] := BOOL_TO_WORD(ADS_Standard.Tags.Status.T_BT1_AL);
GVL.mb_Input_Registers[922] := BOOL_TO_WORD(ADS_Standard.Tags.Status.T_BP1_AL);
GVL.mb_Input_Registers[923] := BOOL_TO_WORD(ADS_Standard.Tags.Status.F_BP1_AL);
GVL.mb_Input_Registers[924] := BOOL_TO_WORD(ADS_Standard.Tags.Status.T_BT1_FAULT);
GVL.mb_Input_Registers[925] := BOOL_TO_WORD(ADS_Standard.Tags.Status.BT1_FAULT);
GVL.mb_Input_Registers[926] := BOOL_TO_WORD(ADS_Standard.Tags.Status.T_BT2_FAULT);
GVL.mb_Input_Registers[927] := BOOL_TO_WORD(ADS_Standard.Tags.Status.T_BT3_FAULT);
GVL.mb_Input_Registers[928] := BOOL_TO_WORD(ADS_Standard.Tags.Status.F_BT1_FAULT);
GVL.mb_Input_Registers[929] := BOOL_TO_WORD(ADS_Standard.Tags.Status.F_BT2_FAULT);
GVL.mb_Input_Registers[930] := BOOL_TO_WORD(ADS_Standard.Tags.Status.BT2_FAULT);
GVL.mb_Input_Registers[931] := BOOL_TO_WORD(ADS_Standard.Tags.Status.H_BT1_FAULT);
GVL.mb_Input_Registers[932] := BOOL_TO_WORD(ADS_Standard.Tags.Status.T_BP1_FAULT);
GVL.mb_Input_Registers[933] := BOOL_TO_WORD(ADS_Standard.Tags.Status.F_BP1_FAULT);
GVL.mb_Input_Registers[934] := BOOL_TO_WORD(ADS_Standard.Tags.Status.T_BP2_FAULT);
GVL.mb_Input_Registers[935] := BOOL_TO_WORD(ADS_Standard.Tags.Status.F_BP2_FAULT);
GVL.mb_Input_Registers[936] := BOOL_TO_WORD(ADS_Standard.Tags.Status.F_BP3_FAULT);
GVL.mb_Input_Registers[937] := BOOL_TO_WORD(ADS_Standard.Tags.Status.T_BR1_AL);
GVL.mb_Input_Registers[938] := BOOL_TO_WORD(ADS_Standard.Tags.Status.F_BR1_AL);
GVL.mb_Input_Registers[939] := BOOL_TO_WORD(ADS_Standard.Tags.Status.T_BF1_FAULT);
GVL.mb_Input_Registers[940] := BOOL_TO_WORD(ADS_Standard.Tags.Status.F_BF1_FAULT);
END_ACTION

END_FUNCTION_BLOCK

// ---- DUTs/IO/TemperatureInput.TcPOU
FUNCTION_BLOCK TemperatureInput EXTENDS AnalogInput
VAR_INPUT
END_VAR
VAR_OUTPUT
END_VAR
VAR
END_VAR
VAR PERSISTENT
END_VAR

SUPER^();
SignedWord := TRUE;

METHOD FB_init : BOOL
VAR_INPUT
	bInitRetains : BOOL; // if TRUE, the retain variables are initialized (warm start / cold start)
	bInCopyCode : BOOL;  // if TRUE, the instance afterwards gets moved into the copy code (online change)
END_VAR
IF bInitRetains THEN
	ProcessMin := -5000;
	ProcessMax := 15000;
	MinValue := -50;
	MaxValue := 150;
END_IF
END_METHOD

END_FUNCTION_BLOCK

// ---- DUTs/IO/AnalogInput.TcPOU
FUNCTION_BLOCK AnalogInput EXTENDS BaseIO
VAR_INPUT
	ProcessValue: LREAL;
	Override: BOOL;
	OverrideValue: LREAL;
END_VAR
VAR_OUTPUT
	Value: LREAL;
END_VAR
VAR
	InitDone: BOOL;
	TempValue: LREAL;
END_VAR
VAR PERSISTENT
	SignedWord: BOOL;
	ProcessMin: DINT := 0;
	ProcessMax: DINT := 16#3FFF;
	MinValue: LREAL := 0;
	MaxValue: LREAL := 1;
	SavedOverride: BOOL;
	SavedOverrideValue: LREAL;
END_VAR

SUPER^();
IF NOT InitDone THEN
	InitDone := TRUE;
	OverrideValue := SavedOverrideValue;
	Override := SavedOverride;	
END_IF
IF NOT Override THEN
	TempValue := ProcessValue;
	IF SignedWord THEN
		IF ProcessValue >= 16#8000 THEN
			TempValue := TempValue - 16#10000;
		END_IF
	END_IF
	Value := GetValue();
	Error := ProcessError;
	ErrorCode := ProcessErrorCode;
ELSE
	Value := OverrideValue;
	Error := FALSE;
	ErrorCode := 0;
END_IF
SavedOverride := Override;
SavedOverrideValue := OverrideValue;

METHOD GetValue : LREAL
VAR_INPUT
END_VAR
GetValue := (LimitValue(TempValue, ProcessMin, ProcessMax) - ProcessMin) / (ProcessMax - ProcessMin) * (MaxValue - MinValue) + MinValue;
END_METHOD

END_FUNCTION_BLOCK

// ---- DUTs/GreenMaster/IO/GreenMasterDO.TcPOU
FUNCTION_BLOCK GreenMasterDO EXTENDS GreenMasterDO_Base
VAR_INPUT
END_VAR
VAR_OUTPUT
END_VAR
VAR_IN_OUT
END_VAR
VAR
	IO_DO_01: DigitalOutput;
	IO_DO_02: DigitalOutput;
	IO_DO_03: DigitalOutput;
	IO_DO_04: DigitalOutput;
	IO_DO_05: DigitalOutput;
	IO_DO_06: DigitalOutput;
	IO_DO_07: DigitalOutput;
	IO_DO_08: DigitalOutput;
	IO_DO_09: DigitalOutput;
	IO_DO_10: DigitalOutput;
	IO_DO_11: DigitalOutput;
	IO_DO_12: DigitalOutput;
	IO_DO_13: DigitalOutput;
	IO_DO_14: DigitalOutput;
	IO_RDO_01: DigitalOutput;
	IO_RDO_02: DigitalOutput;
	IO_RDO_03: DigitalOutput;
	IO_RDO_04: DigitalOutput;
	IO_DO_16: DigitalOutput;
END_VAR


// PAGE Digital outputs
IO_DO_01(Value := H_GP1); // DigitalOutput
IO_DO_02(Value := C_GP1); // DigitalOutput
DOut.DO01 := IO_DO_01.ProcessValue;
DOut.DO02 := IO_DO_02.ProcessValue;
IO_DO_03(Value := ExhaustRunning); // DigitalOutput
IO_DO_04(Value := F_QM1); // DigitalOutput
DOut.DO03 := IO_DO_03.ProcessValue;
DOut.DO04 := IO_DO_04.ProcessValue;
IO_DO_05(Value := T_QM2); // DigitalOutput
IO_DO_06(Value := R_QM1); // DigitalOutput
DOut.DO05 := IO_DO_05.ProcessValue;
DOut.DO06 := IO_DO_06.ProcessValue;
IO_DO_07(Value := F_QM2); // DigitalOutput
IO_DO_08(Value := SupplyRunning); // DigitalOutput
DOut.DO07 := IO_DO_07.ProcessValue;
DOut.DO08 := IO_DO_08.ProcessValue;
IO_DO_09(Value := T_QM1_1); // DigitalOutput
IO_DO_10(Value := T_QM1_2); // DigitalOutput
DOut.DO09 := IO_DO_09.ProcessValue;
DOut.DO10 := IO_DO_10.ProcessValue;
IO_DO_11(Value := T_QM1_3); // DigitalOutput
IO_DO_12(Value := T_QM1_4); // DigitalOutput
DOut.DO11 := IO_DO_11.ProcessValue;
DOut.DO12 := IO_DO_12.ProcessValue;
IO_DO_13(Value := T_QM1_5); // DigitalOutput
IO_DO_14(Value := T_QM1_6); // DigitalOutput
DOut.DO13 := IO_DO_13.ProcessValue;
DOut.DO14 := IO_DO_14.ProcessValue;
IO_DO_16(Value := P2); // DigitalOutput
DOut.DO16 := IO_DO_16.ProcessValue;

// PAGE Relay outputs
IO_RDO_01(Value := AlarmRelayA); // DigitalOutput
Globals.IO.DOut.RDO01 := IO_RDO_01.ProcessValue;
IO_RDO_02(Value := AlarmRelayB); // DigitalOutput
Globals.IO.DOut.RDO02 := IO_RDO_02.ProcessValue;
IO_RDO_03(Value := AlarmRelayC); // DigitalOutput
Globals.IO.DOut.RDO03 := IO_RDO_03.ProcessValue;
IO_RDO_04(Value := AlarmRelayD); // DigitalOutput
Globals.IO.DOut.RDO04 := IO_RDO_04.ProcessValue;

METHOD SetOverrides : BOOL
VAR_INPUT
	Override: DigitalOutputOverrideParameters;
END_VAR
IF Main.ManualAllowed THEN
	IO_DO_01.Override := Override.H_GP1_Override;
	IO_DO_01.OverrideValue := Override.H_GP1_OverrideValue;
	IO_DO_02.Override := Override.C_GP1_Override;
	IO_DO_02.OverrideValue := Override.C_GP1_OverrideValue;
	IO_DO_03.Override := Override.F_RUN_Override;
	IO_DO_03.OverrideValue := Override.F_RUN_OverrideValue;
	IO_DO_04.Override := Override.F_QM1_Override;
	IO_DO_04.OverrideValue := Override.F_QM1_OverrideValue;
	IO_DO_05.Override := Override.T_QM2_Override;
	IO_DO_05.OverrideValue := Override.T_QM2_OverrideValue;
	IO_DO_06.Override := Override.R_QM1_Override;
	IO_DO_06.OverrideValue := Override.R_QM1_OverrideValue;
	IO_DO_07.Override := Override.F_QM2_Override;
	IO_DO_07.OverrideValue := Override.F_QM2_OverrideValue;
	IO_DO_08.Override := Override.T_RUN_Override;
	IO_DO_08.OverrideValue := Override.T_RUN_OverrideValue;
	IO_DO_09.Override := Override.T_QM1_1_Override;
	IO_DO_09.OverrideValue := Override.T_QM1_1_OverrideValue;
	IO_DO_10.Override := Override.T_QM1_2_Override;
	IO_DO_10.OverrideValue := Override.T_QM1_2_OverrideValue;
	IO_DO_11.Override := Override.T_QM1_3_Override;
	IO_DO_11.OverrideValue := Override.T_QM1_3_OverrideValue;
	IO_DO_12.Override := Override.T_QM1_4_Override;
	IO_DO_12.OverrideValue := Override.T_QM1_4_OverrideValue;
	IO_DO_13.Override := Override.T_QM1_5_Override;
	IO_DO_13.OverrideValue := Override.T_QM1_5_OverrideValue;
	IO_DO_14.Override := Override.T_QM1_6_Override;
	IO_DO_14.OverrideValue := Override.T_QM1_6_OverrideValue;
	IO_DO_16.Override := Override.P2_Override;
	IO_DO_16.OverrideValue := Override.P2_OverrideValue;
ELSE	
	IO_DO_01.Override := FALSE;
	IO_DO_02.Override := FALSE;
	IO_DO_03.Override := FALSE;
	IO_DO_04.Override := FALSE;
	IO_DO_05.Override := FALSE;
	IO_DO_06.Override := FALSE;
	IO_DO_07.Override := FALSE;
	IO_DO_08.Override := FALSE;
	IO_DO_09.Override := FALSE;
	IO_DO_10.Override := FALSE;
	IO_DO_11.Override := FALSE;
	IO_DO_12.Override := FALSE;
	IO_DO_13.Override := FALSE;
	IO_DO_14.Override := FALSE;
	IO_DO_16.Override := FALSE;
END_IF
END_METHOD

END_FUNCTION_BLOCK

// ---- DUTs/GreenMaster/IO/GreenMasterAO.TcPOU
FUNCTION_BLOCK GreenMasterAO EXTENDS GreenMasterAO_Base
VAR_INPUT
END_VAR
VAR_OUTPUT
END_VAR
VAR
	IO_AO_01: AnalogOutput;	
	IO_AO_02: AnalogOutput;	
	IO_AO_03: AnalogOutput;	
	IO_AO_04: AnalogOutput;	
	IO_AO_05: AnalogOutput;	
END_VAR


// PAGE AO
IO_AO_01(Value := F_QN1); // AnalogOutput
AOut.AO01 := LREAL_TO_WORD(IO_AO_01.ProcessValue);
IO_AO_02(Value := T_GQ1); // AnalogOutput
AOut.AO02 := LREAL_TO_WORD(IO_AO_02.ProcessValue);
IO_AO_03(Value := F_GQ1); // AnalogOutput
AOut.AO03 := LREAL_TO_WORD(IO_AO_03.ProcessValue);
IO_AO_04(Value := C_QN1); // AnalogOutput
AOut.AO04 := LREAL_TO_WORD(IO_AO_04.ProcessValue);
IO_AO_05(Value := H_QN1); // AnalogOutput
AOut.AO05 := LREAL_TO_WORD(IO_AO_05.ProcessValue);

METHOD SetOverrideC_QN1 : BOOL
VAR_INPUT
	Override: BOOL;
	OverrideValue: LREAL;
	Parameters: REFERENCE TO GreenMasterBaseParameters;
END_VAR
IO_AO_04.SetOverride2(OverrideIN := Override,
	OverrideValueIN := OverrideValue);
END_METHOD

METHOD SetOverrideF_GQ1 : BOOL
VAR_INPUT
	Override: BOOL;
	OverrideValue: LREAL;
	Parameters: REFERENCE TO GreenMasterBaseParameters;
END_VAR
IO_AO_03.SetOverride2(OverrideIN := Override, OverrideValueIN := OverrideValue);
END_METHOD

METHOD SetOverrideF_QN1 : BOOL
VAR_INPUT
	Override: BOOL;
	OverrideValue: LREAL;
	Parameters: REFERENCE TO GreenMasterBaseParameters;
END_VAR
IO_AO_01.SetOverride2(OverrideIN := Override, OverrideValueIN := OverrideValue);
END_METHOD

METHOD SetOverrideH_QN1 : BOOL
VAR_INPUT
	Override: BOOL;
	OverrideValue: LREAL;
	Parameters: REFERENCE TO GreenMasterBaseParameters;
END_VAR
IO_AO_05.SetOverride2(OverrideIN := Override, OverrideValueIN := OverrideValue);
END_METHOD

METHOD SetOverrideT_GQ1 : BOOL
VAR_INPUT
	Override: BOOL;
	OverrideValue: LREAL;
	Parameters: REFERENCE TO GreenMasterBaseParameters;
END_VAR
IO_AO_02.SetOverride2(OverrideIN := Override, OverrideValueIN := OverrideValue);
END_METHOD

END_FUNCTION_BLOCK

// ---- DUTs/IO/AnalogOutput.TcPOU
FUNCTION_BLOCK AnalogOutput EXTENDS BaseIO
VAR_INPUT
	Value: LREAL;
	Override: BOOL;
	OverrideValue: LREAL;
END_VAR
VAR_OUTPUT
	ProcessValue: LREAL;
	ValueOut: LREAL;
END_VAR
VAR
	InitDone: BOOL;
	TempValue: LREAL;
	OutValue: LREAL;
	Override2: BOOL;
	OverrideValue2: LREAL;
END_VAR
VAR PERSISTENT
	SignedWord: BOOL;
	ProcessMin: DINT := 0;
	ProcessMax: DINT := 16#7FFF;
	MinValue: LREAL := 0;
	MaxValue: LREAL := 1;
	SavedOverride: BOOL;
	SavedOverrideValue: LREAL;
	SavedOverride2: BOOL;
	SavedOverrideValue2: LREAL;
END_VAR

SUPER^();
IF NOT InitDone THEN
	InitDone := TRUE;
	OverrideValue := SavedOverrideValue;
	Override := SavedOverride;	
	OverrideValue2 := SavedOverrideValue2;
	Override2 := SavedOverride2;	
END_IF
TempValue := Value;
IF Override2 THEN
	TempValue := OverrideValue2;
END_IF
IF Override THEN
	TempValue := OverrideValue;
END_IF
OutValue := (LimitValue(TempValue, MinValue, MaxValue) - MinValue) / (MaxValue - MinValue) * (ProcessMax - ProcessMin) + ProcessMin;
IF SignedWord THEN
	IF OutValue < 0 THEN
		OutValue := OutValue + 16#10000;
	END_IF
END_IF
ProcessValue := OutValue;
SavedOverride := Override;
SavedOverrideValue := OverrideValue;
SavedOverride2 := Override2;
SavedOverrideValue2 := OverrideValue2;
ValueOut :=TempValue;

METHOD SetOverride2 : BOOL
VAR_INPUT
	OverrideIN: BOOL;
	OverrideValueIN: LREAL;
END_VAR
Override2 := OverrideIN;
OverrideValue2 := OverrideValueIN;
END_METHOD

END_FUNCTION_BLOCK

// ---- DUTs/Utilities/REAL_TO_WORD_SAFE.TcPOU
FUNCTION REAL_TO_WORD_SAFE : WORD
VAR_INPUT
	Value: REAL;
END_VAR
VAR
END_VAR

REAL_TO_WORD_SAFE := TO_WORD(TO_INT(Value));

END_FUNCTION

// ---- DUTs/Custom/ExtraAlarms/ExtraAlarms_Interface.TcPOU
FUNCTION_BLOCK ExtraAlarms_Interface
VAR_INPUT
	EN: BOOL;
END_VAR
VAR_OUTPUT
	ENO: BOOL;
END_VAR
VAR
	InitDone: BOOL;
	Parameters: REFERENCE TO GreenMasterBaseParameters;
END_VAR

IF NOT InitDone THEN
	Parameters REF= Main.GreenMaster.GetParameters();
	InitDone := TRUE;
END_IF;

ENO := EN;

IF EN THEN
	// Status transfers
	ADS_ExtraAlarms.Tags.Status.EXTRA_01_AL := Parameters.Alarm.Active.A.AL01;
	ADS_ExtraAlarms.Tags.Status.EXTRA_02_AL := Parameters.Alarm.Active.A.AL02;
	ADS_ExtraAlarms.Tags.Status.EXTRA_03_AL := Parameters.Alarm.Active.A.AL03;
	ADS_ExtraAlarms.Tags.Status.EXTRA_04_AL := Parameters.Alarm.Active.A.AL04;
	ADS_ExtraAlarms.Tags.Status.EXTRA_05_AL := Parameters.Alarm.Active.A.AL05;
	ADS_ExtraAlarms.Tags.Status.EXTRA_06_AL := Parameters.Alarm.Active.A.AL06;
	ADS_ExtraAlarms.Tags.Status.EXTRA_07_AL := Parameters.Alarm.Active.A.AL07;
	ADS_ExtraAlarms.Tags.Status.EXTRA_08_AL := Parameters.Alarm.Active.A.AL08;
END_IF

END_FUNCTION_BLOCK

// ---- DUTs/Custom/SmokeControl/SmokeControl_Interface.TcPOU
FUNCTION_BLOCK SmokeControl_Interface
VAR_INPUT
	EN: BOOL;
END_VAR
VAR_OUTPUT
	ENO: BOOL;
END_VAR
VAR
	InitDone: BOOL;
	Parameters: REFERENCE TO GreenMasterBaseParameters;
	ParametersSC: REFERENCE TO SmokeControlParametersBase;
END_VAR

IF NOT InitDone THEN
	Parameters REF= Main.GreenMaster.GetParameters();
	ParametersSC REF= Main.GreenMaster.GetParametersSC();
	InitDone := TRUE;
END_IF;

ENO := EN;

IF EN THEN
	// Status
	ADS_SmokeControl.Tags.Status.COMM_AL := (ParametersSC.DamperModules.Unit01.EN AND ParametersSC.DamperModules.Unit01.Error) OR
		(ParametersSC.DamperModules.Unit02.EN AND ParametersSC.DamperModules.Unit02.Error) OR
		(ParametersSC.DamperModules.Unit03.EN AND ParametersSC.DamperModules.Unit03.Error) OR
		(ParametersSC.DamperModules.Unit04.EN AND ParametersSC.DamperModules.Unit04.Error) OR
		(ParametersSC.DamperModules.Unit05.EN AND ParametersSC.DamperModules.Unit05.Error) OR
		(ParametersSC.DamperModules.Unit06.EN AND ParametersSC.DamperModules.Unit06.Error) OR
		(ParametersSC.DamperModules.Unit07.EN AND ParametersSC.DamperModules.Unit07.Error) OR
		(ParametersSC.DamperModules.Unit08.EN AND ParametersSC.DamperModules.Unit08.Error) OR
		(ParametersSC.DamperModules.Unit09.EN AND ParametersSC.DamperModules.Unit09.Error) OR
		(ParametersSC.DamperModules.Unit10.EN AND ParametersSC.DamperModules.Unit10.Error) OR
		(ParametersSC.DamperModules.Unit11.EN AND ParametersSC.DamperModules.Unit11.Error) OR
		(ParametersSC.DamperModules.Unit12.EN AND ParametersSC.DamperModules.Unit12.Error) OR
		(ParametersSC.DamperModules.Unit13.EN AND ParametersSC.DamperModules.Unit13.Error) OR
		(ParametersSC.DamperModules.Unit14.EN AND ParametersSC.DamperModules.Unit14.Error) OR
		(ParametersSC.DamperModules.Unit15.EN AND ParametersSC.DamperModules.Unit15.Error);
	UpdateModuleTags(ADS_SmokeControl.Tags.Status.UNIT_01, ParametersSC.DamperModules.Unit01);
	UpdateModuleTags(ADS_SmokeControl.Tags.Status.UNIT_02, ParametersSC.DamperModules.Unit02);
	UpdateModuleTags(ADS_SmokeControl.Tags.Status.UNIT_03, ParametersSC.DamperModules.Unit03);
	UpdateModuleTags(ADS_SmokeControl.Tags.Status.UNIT_04, ParametersSC.DamperModules.Unit04);
	UpdateModuleTags(ADS_SmokeControl.Tags.Status.UNIT_05, ParametersSC.DamperModules.Unit05);
	UpdateModuleTags(ADS_SmokeControl.Tags.Status.UNIT_06, ParametersSC.DamperModules.Unit06);
	UpdateModuleTags(ADS_SmokeControl.Tags.Status.UNIT_07, ParametersSC.DamperModules.Unit07);
	UpdateModuleTags(ADS_SmokeControl.Tags.Status.UNIT_08, ParametersSC.DamperModules.Unit08);
	UpdateModuleTags(ADS_SmokeControl.Tags.Status.UNIT_09, ParametersSC.DamperModules.Unit09);
	UpdateModuleTags(ADS_SmokeControl.Tags.Status.UNIT_10, ParametersSC.DamperModules.Unit10);
	UpdateModuleTags(ADS_SmokeControl.Tags.Status.UNIT_11, ParametersSC.DamperModules.Unit11);
	UpdateModuleTags(ADS_SmokeControl.Tags.Status.UNIT_12, ParametersSC.DamperModules.Unit12);
	UpdateModuleTags(ADS_SmokeControl.Tags.Status.UNIT_13, ParametersSC.DamperModules.Unit13);
	UpdateModuleTags(ADS_SmokeControl.Tags.Status.UNIT_14, ParametersSC.DamperModules.Unit14);
	UpdateModuleTags(ADS_SmokeControl.Tags.Status.UNIT_15, ParametersSC.DamperModules.Unit15);
END_IF

METHOD UpdateModuleTags : BOOL
VAR_INPUT
	SxDuoInterface: REFERENCE TO SxDuoInterface;
	SxDuoUnit: reference to SxDuoUnit;
END_VAR
SxDuoInterface.TEXT_PV := SxDuoUnit.Text_CP1252;
SxDuoInterface.DAMPER1_AL := SxDuoUnit.SxDuoStatus.Damper1Alarm;
SxDuoInterface.DAMPER2_AL := SxDuoUnit.SxDuoStatus.Damper2Alarm;
SxDuoInterface.DAMPER1_V0 := SxDuoUnit.SxDuoStatus.Damper1Closed;
SxDuoInterface.DAMPER2_V0 := SxDuoUnit.SxDuoStatus.Damper2Closed;
SxDuoInterface.DAMPER1_V1 := SxDuoUnit.SxDuoStatus.Damper1Open;
SxDuoInterface.DAMPER2_V1 := SxDuoUnit.SxDuoStatus.Damper2Open;
SxDuoInterface.EXERCISING_V := SxDuoUnit.SxDuoStatus.Exercising;
SxDuoInterface.FIRE_AL := SxDuoUnit.SxDuoStatus.FireAlarm;
SxDuoInterface.FIRE_FAULT := SxDuoUnit.SxDuoStatus.ServiceAlarm;
SxDuoInterface.COMM_FAULT := SxDuoUnit.Error;
END_METHOD

END_FUNCTION_BLOCK

// ---- DUTs/Custom/Redundancy/Redundancy.TcPOU
FUNCTION_BLOCK Redundancy
VAR_INPUT
	EN: BOOL;
	_UPPSTART_DONE:BOOL;
	_TF_CMD:BOOL;
	_TF_V:BOOL;
	_TF_OP:REAL;
	_TL_GP_PV:REAL;
	_FF_CMD:BOOL;
	_FF_V:BOOL;
	_FF_OP:REAL;
	_FL_GP_PV:REAL;
	_SERVICEBRYTARE:BOOL;
	
	_B_AMSID:STRING;
	_B_VARIABLE:STRING;
END_VAR
VAR_OUTPUT
	ENO: BOOL;	
END_VAR
VAR
	Parameters: REFERENCE TO GreenMasterBaseParametersFB;
	GM_XXL: REFERENCE TO GreenMasterXXL_FB;
	
	B_STATUS:adsValue_AggStat;		// Det andra aggregatet
	A_STATUS:AggStat;				// Detta aggregatet

END_VAR
VAR_INPUT PERSISTENT
	AGG_A:BOOL;	// True = A false = B
END_VAR

(*
Samdrift av LB01 och LB02. En- till tvåaggregatsdrift och två- till enaggregatsdrift
då optimalt luftflöde överskrids resp. underskrids med 3% av
aggregatens totala luftflöde i inställd tid. Efter att båda aggregaten tagits i drift
skall de, efter inställd tid, regleras parallellt på samma signal så att pendlingar i
systemen begränsas.
Drifttidsutjämning genom att veckovis rotera första- resp. andraaggregat.
*)
IF EN THEN
	// Fyll i Aggregatstatus till redundant aggregat
	A_STATUS.Driftfel 	:= _UPPSTART_DONE AND ((_TF_CMD AND NOT _TF_V) OR (_FF_CMD AND NOT _FF_V));	// Uppstart klar och driftfel TF eller FF (Innan larmtid)
	A_STATUS.FF_OP 		:= _FF_OP;//FO2._orderOp;
	A_STATUS.FF_CMD 	:= _FF_CMD;
	A_STATUS.GP11_PV 	:= _TL_GP_PV;
	A_STATUS.GP12_PV 	:= _FL_GP_PV;
	A_STATUS.SO1 		:= _SERVICEBRYTARE;
//	A_STATUS.ST_OP 		:= ST22.OP;
	A_STATUS.TF_OP 		:= _TF_OP;
	A_STATUS.TF_CMD 	:= _TF_CMD;

	// Hämta aggregatstatus från redundant aggregat
	B_STATUS.AMSID:=_B_AMSID;//'5.83.130.125.1.1';
	B_STATUS.AMSPORT:=851;
	B_STATUS.VARIABLE:=_B_VARIABLE;//'GF_5000_5078.p05.B.B_STATUS';
	B_STATUS();

	// --------------------------------------------------------------------------------
	// Transfer from Redundancy to settings

	// Status transfers
//	GVL_Redundancy.Tags.Status.FF_CMD := GM_XXL.SupplyFanControl.ENO;
	
	// Tillfällig lösning
	// Set AMSID
	
END_IF

END_FUNCTION_BLOCK

// ---- DUTs/Custom/Redundancy/adsValue_AggStat.TcPOU
FUNCTION_BLOCK adsValue_AggStat
VAR_INPUT
	_r_tsNow:TIMESTRUCT;		(* Aktuell tid *)
END_VAR
VAR_OUTPUT
	SO1:BOOL;		// Serviceomkopplarläge 1 = service
	Driftfel:BOOL;	// Aggregatet är i driftfel eller
	TF_OP:REAL;		// Utsignal tilluftsfläkt
	TF_CMD:BOOL;	// Manöver tilluftsflöäkt
	FF_CMD:BOOL;	// Manöver tilluftsflöäkt	
	FF_OP:REAL;		// Utsignal frånluftsfläkt
	ST_OP:REAL;		// Utsignal Till- och frånluftsspjäll
	GP11_PV:REAL;
	GP11_FAULT:BOOL;
	GP12_PV:REAL;
	GP12_FAULT:BOOL;
	FAULT:BOOL;		(* [type=DIGITAL], [scale=|||], [descr=Kommunikationsfel], [format=#], [engunit=], [prio=<givarfelprio>], [setting=] *)
END_VAR
VAR
	ReadAdsSymbol:FB_ReadAdsSymByName;
	_Data:AggStat;
	_ton:TON;
END_VAR
VAR_INPUT PERSISTENT
	AMSID:STRING;			(* [rename=AMSID:SP1], [type=STRING], [scale=|||], [descr=AMS-Net-ID], [format=], [engunit=], [prio=], [setting=1] *)
	AMSPORT:UINT:=851;		(* [rename=AMSPORT:SP2], [type=STRING], [scale=|||], [descr=AMS-Net-Port], [format=], [engunit=], [prio=], [setting=1] *)
	VARIABLE:STRING;		(* [rename=AMSID:SP3], [type=STRING], [scale=|||], [descr=Variabelnamn], [format=], [engunit=], [prio=], [setting=1] *)
	iLastSec:INT;
END_VAR
(* Summalarm *)
VAR_INPUT
	_SLPRIO:INT:=3;
END_VAR

//	_ton(IN:=NOT _ton.Q, PT:=T#100MS);
	IF NOT ReadAdsSymbol.bBusy THEN// _ton.Q THEN
		ReadAdsSymbol(	bRead		:=	TRUE,
						sNetId		:=	AMSID,
						nPort		:=	AMSPORT,
						sVarName	:=	VARIABLE,
						nDestAddr	:=	ADR(_Data),
						nLen		:=	SIZEOF(AggStat),
						tTimeout	:=	DEFAULT_ADS_TIMEOUT,
						eComMode	:=	eAdsComModeFastCom);
	END_IF;

	ReadAdsSymbol(	bRead:=FALSE);

	SO1 		:= 	_Data.SO1;
	Driftfel 	:= 	_Data.Driftfel;
	TF_OP		:=	_Data.TF_OP;
	TF_CMD		:=	_Data.TF_CMD;
	FF_OP		:=	_Data.FF_OP;
	FF_CMD		:=	_Data.FF_CMD;
	ST_OP		:=	_Data.ST_OP;
	GP11_PV		:=	_Data.GP11_PV;
	GP11_FAULT	:=	_Data.GP11_FAULT;
	GP12_PV		:=	_Data.GP12_PV;	
	GP12_FAULT	:=	_Data.GP12_FAULT;
	
	FAULT :=ReadAdsSymbol.bError;

	(* Summalarm *)
//	IF  FAULT THEN
//		CASE _SLPRIO OF
//			1: GVL_JITEA._SUMLA_A := TRUE;
//			2: GVL_JITEA._SUMLA_B := TRUE;
//			3: GVL_JITEA._SUMLA_C := TRUE;
//		END_CASE
//	END_IF

END_FUNCTION_BLOCK

// ---- DUTs/GreenMaster/IO/GreenMasterDI.TcPOU
FUNCTION_BLOCK GreenMasterDI EXTENDS GreenMasterDI_Base
VAR_INPUT
END_VAR
VAR_OUTPUT
END_VAR
VAR
	IO_DI_01: DigitalInput;
	IO_DI_02: DigitalInput;
	IO_DI_03: DigitalInput;
	IO_DI_04: DigitalInput;
	IO_DI_05: DigitalInput;
	IO_DI_06: DigitalInput;
	IO_DI_07: DigitalInput;
	IO_DI_08: DigitalInput;
	IO_DI_09: DigitalInput;
	IO_DI_10: DigitalInput;
	IO_DI_11: DigitalInput;
	IO_DI_12: DigitalInput;
	IO_DI_13: DigitalInput;
	IO_DI_14: DigitalInput;
	IO_DI_15: DigitalInput;
	IO_DI_16: DigitalInput;
	IO_DI_17: DigitalInput;
	IO_DI_18: DigitalInput;
	IO_DI_19: DigitalInput;
	IO_DI_20: DigitalInput;
	IO_DI_21: DigitalInput;
	IO_DI_22: DigitalInput;
	IO_DI_23: DigitalInput;
	IO_DI_24: DigitalInput;
	IO_DI_25: DigitalInput;
	IO_DI_26: DigitalInput;
	IO_DI_27: DigitalInput;
	IO_DI_28: DigitalInput;
	IO_DI_29: DigitalInput;
END_VAR


// PAGE Digital Inputs DIXX in Globals are connected to physical inputs
IO_DI_01(ProcessValue := DIn.DI01, Inverted := DInLevels.DI01); // DigitalInput
Auto := IO_DI_01.Value;
IO_DI_02(ProcessValue := DIn.DI02, Inverted := DInLevels.DI02); // DigitalInput
FireExtractAlarm := IO_DI_02.Value;
IO_DI_03(ProcessValue := DIn.DI03, Inverted := DInLevels.DI03); // DigitalInput
FuseAlarm := IO_DI_03.Value;
IO_DI_04(ProcessValue := DIn.DI04, Inverted := DInLevels.DI04); // DigitalInput
Hand := IO_DI_04.Value;
IO_DI_05(ProcessValue := DIn.DI05, Inverted := DInLevels.DI05); // DigitalInput
T_GQ1_Alarm := IO_DI_05.Value;
IO_DI_06(ProcessValue := DIn.DI06, Inverted := DInLevels.DI06); // DigitalInput
F_GQ1_Alarm := IO_DI_06.Value;
IO_DI_07(ProcessValue := DIn.DI07, Inverted := DInLevels.DI07); // DigitalInput
F_QM2_Closed := IO_DI_07.Value;
IO_DI_08(ProcessValue := DIn.DI08, Inverted := DInLevels.DI08); // DigitalInput
F_QM2_Open := IO_DI_08.Value;
IO_DI_09(ProcessValue := DIn.DI09, Inverted := DInLevels.DI09); // DigitalInput
ExtendedOperation := IO_DI_09.Value;
IO_DI_10(ProcessValue := DIn.DI10, Inverted := DInLevels.DI10); // DigitalInput
ServiceAlarmCentralAndSmokeExhaustAir := IO_DI_10.Value;
IO_DI_11(ProcessValue := DIn.DI11, Inverted := DInLevels.DI11); // DigitalInput
FireSupplyAlarm := IO_DI_11.Value;
IO_DI_12(ProcessValue := DIn.DI12, Inverted := DInLevels.DI12); // DigitalInput
ServiceAlarmSupplyAir := IO_DI_12.Value;
IO_DI_13(ProcessValue := DIn.DI13, Inverted := DInLevels.DI13); // DigitalInput
H_GP1_Running := IO_DI_13.Value;
IO_DI_14(ProcessValue := DIn.DI14, Inverted := DInLevels.DI14); // DigitalInput
C_GP1_Running := IO_DI_14.Value;
IO_DI_15(ProcessValue := DIn.DI15, Inverted := DInLevels.DI15); // DigitalInput
TX1_Running := IO_DI_15.Value;
P2_Alarm := IO_DI_23.Value;
IO_DI_16(ProcessValue := DIn.DI16, Inverted := DInLevels.DI16); // DigitalInput
ResetAlarm := IO_DI_16.Value;
IO_DI_17(ProcessValue := DIn.DI17, Inverted := DInLevels.DI17); // DigitalInput
IO_DI_18(ProcessValue := DIn.DI18, Inverted := DInLevels.DI18); // DigitalInput
IO_DI_19(ProcessValue := DIn.DI19, Inverted := DInLevels.DI19); // DigitalInput
IO_DI_20(ProcessValue := DIn.DI20, Inverted := DInLevels.DI20); // DigitalInput
IO_DI_21(ProcessValue := DIn.DI21, Inverted := DInLevels.DI21); // DigitalInput
IO_DI_24(ProcessValue := DIn.DI24, Inverted := DInLevels.DI24); // DigitalInput
IO_DI_22(ProcessValue := DIn.DI22, Inverted := DInLevels.DI22); // DigitalInput
ExpansionVesselAlarm := IO_DI_24.Value;
P2_Running := IO_DI_22.Value;
IO_DI_23(ProcessValue := DIn.DI23, Inverted := DInLevels.DI23); // DigitalInput
IO_DI_25(ProcessValue := DIn.DI25, Inverted := DInLevels.DI25); // DigitalInput
FireActivateSupplyAir := IO_DI_25.Value;
IO_DI_26(ProcessValue := DIn.DI26, Inverted := DInLevels.DI26); // DigitalInput
FireDeactivateSupplyAir := IO_DI_26.Value;
IO_DI_27(ProcessValue := DIn.DI27, Inverted := DInLevels.DI27); // DigitalInput
FireActivateExtractAir := IO_DI_27.Value;
IO_DI_28(ProcessValue := DIn.DI28, Inverted := DInLevels.DI28); // DigitalInput
IO_DI_29(ProcessValue := DIn.DI29, Inverted := DInLevels.DI29); // DigitalInput
FireDeactivateExtractAir := IO_DI_28.Value;
F_QM1_Closed := IO_DI_20.Value;
F_QM1_Open := IO_DI_21.Value;
T_QM2_Closed := IO_DI_18.Value;
T_QM2_Open := IO_DI_19.Value;

END_FUNCTION_BLOCK

// ---- DUTs/GreenMaster/IO/GreenMasterAI.TcPOU
FUNCTION_BLOCK GreenMasterAI EXTENDS GreenMasterAI_Base
VAR_INPUT
END_VAR
VAR_OUTPUT
END_VAR
VAR
	IO_AI_01: TemperatureInput;
	IO_AI_02: TemperatureInput;
	IO_AI_03: TemperatureInput;
	IO_AI_04: TemperatureInput;
	IO_AI_05: TemperatureInput;
	IO_AI_06: TemperatureInput;
	IO_AI_07: TemperatureInput;
	IO_AI_08: TemperatureInput;
END_VAR


// PAGE AI
IO_AI_01(ProcessError := AIn.AI01_Error, ProcessValue := AIn.AI01); // TemperatureInput
F_BT1_Error := IO_AI_01.Error;
IO_AI_02(ProcessError := AIn.AI02_Error, ProcessValue := AIn.AI02); // TemperatureInput
F_BT1 := IO_AI_01.Value;
T_BT2_Error := IO_AI_02.Error;
T_BT2 := IO_AI_02.Value;
IO_AI_03(ProcessError := AIn.AI03_Error, ProcessValue := AIn.AI03); // TemperatureInput
T_BT3_Error := IO_AI_03.Error;
IO_AI_04(ProcessError := AIn.AI04_Error, ProcessValue := AIn.AI04); // TemperatureInput
T_BT3 := IO_AI_03.Value;
H_BT1_Error := IO_AI_04.Error;
H_BT1 := IO_AI_04.Value;
IO_AI_05(ProcessError := AIn.AI05_Error, ProcessValue := AIn.AI05); // TemperatureInput
T_BT1_Error := IO_AI_05.Error;
IO_AI_06(ProcessError := AIn.AI06_Error, ProcessValue := AIn.AI06); // TemperatureInput
T_BT1 := IO_AI_05.Value;
BT1_Error := IO_AI_06.Error;
BT1 := IO_AI_06.Value;
IO_AI_07(ProcessError := AIn.AI07_Error, ProcessValue := AIn.AI07); // TemperatureInput
BT2_Error := IO_AI_07.Error;
IO_AI_08(ProcessError := AIn.AI08_Error, ProcessValue := AIn.AI08); // TemperatureInput
BT2 := IO_AI_07.Value;
F_BT2_Error := IO_AI_08.Error;
F_BT2 := IO_AI_08.Value;

END_FUNCTION_BLOCK

// ---- DUTs/GreenMaster/IO/GreenMasterAIU_ModbusRTU.TcPOU
FUNCTION_BLOCK GreenMasterAIU_ModbusRTU EXTENDS GreenMasterAIU_Base
VAR_IN_OUT
	Parameters:GreenMasterBaseParameters;
END_VAR
VAR_OUTPUT
END_VAR
VAR
	ModbusRTU: ModbusRTU;
	ModbusWord_T_BF1: ModbusReadWord;
	ModbusWord_F_BF1: ModbusReadWord;
	ModbusWord_T_BP1: ModbusReadWord;
	ModbusWord_F_BP1: ModbusReadWord;
	ModbusWord_T_BP2: ModbusReadWord;
	ModbusWord_F_BP2: ModbusReadWord;
	ModbusWord_F_BP3: ModbusReadWord;
	IO_AI_T_BP1: PressureInput;	

	IO_AI_F_BP1: PressureInput;
	IO_AI_T_BP2: PressureInput;
	IO_AI_F_BP2: PressureInput;
	IO_AI_F_BP3: PressureInput;
	IO_AI_T_BF1: FlowInput;
	IO_AI_F_BF1: FlowInput;
	EBM_Power_0: EBM_Power;
	EBM_Power_1: EBM_Power;
	Gebhardt_Power_0: Gebhardt_Power;
	Gebhardt_Power_1: Gebhardt_Power;
	EBM_Speed_0: EBM_Speed;
	EBM_Speed_1: EBM_Speed;
	Gebhardt_Speed_0: Gebhardt_Speed;
	Gebhardt_Speed_1: Gebhardt_Speed;
END_VAR
VAR // added by the converter: edge detectors and wires of the graphical bodies
    _w1 : ANY;
END_VAR


// PAGE Pressure inputs
ModbusRTU(EN := EN);
ModbusWord_T_BF1(
    EN := ModbusRTU.ENO,
    Modbus := ModbusRTU,
    UnitID := 114,
    RegisterType := ModbusRegisterType.InputRegister,
    Register := 1); // ModbusReadWord
T_BF1_Error := IO_AI_T_BF1.Error;
T_BF1 := IO_AI_T_BF1.Value;
ModbusWord_F_BF1(
    EN := ModbusRTU.ENO,
    Modbus := ModbusRTU,
    UnitID := 113,
    RegisterType := ModbusRegisterType.InputRegister,
    Register := 1); // ModbusReadWord
F_BF1_Error := IO_AI_F_BF1.Error;
F_BF1 := IO_AI_F_BF1.Value;
ModbusWord_T_BP1(
    EN := ModbusRTU.ENO,
    Modbus := ModbusRTU,
    UnitID := 115,
    RegisterType := ModbusRegisterType.InputRegister,
    Register := 1); // ModbusReadWord
T_BP1_Error := IO_AI_T_BP1.Error;
T_BP1 := IO_AI_T_BP1.Value;
ModbusWord_F_BP1(
    EN := ModbusRTU.ENO,
    Modbus := ModbusRTU,
    UnitID := 110,
    RegisterType := ModbusRegisterType.InputRegister,
    Register := 1); // ModbusReadWord
F_BP1_Error := IO_AI_F_BP1.Error;
F_BP1 := IO_AI_F_BP1.Value;
ModbusWord_T_BP2(
    EN := ModbusRTU.ENO,
    Modbus := ModbusRTU,
    UnitID := 116,
    RegisterType := ModbusRegisterType.InputRegister,
    Register := 1); // ModbusReadWord
T_BP2_Error := IO_AI_T_BP2.Error;
T_BP2 := IO_AI_T_BP2.Value;
ModbusWord_F_BP2(
    EN := ModbusRTU.ENO,
    Modbus := ModbusRTU,
    UnitID := 111,
    RegisterType := ModbusRegisterType.InputRegister,
    Register := 1); // ModbusReadWord
F_BP2_Error := IO_AI_F_BP2.Error;
F_BP2 := IO_AI_F_BP2.Value;
ModbusWord_F_BP3(
    EN := ModbusRTU.ENO,
    Modbus := ModbusRTU,
    UnitID := 112,
    RegisterType := ModbusRegisterType.InputRegister,
    Register := 1); // ModbusReadWord
F_BP3_Error := IO_AI_F_BP3.Error;
F_BP3 := IO_AI_F_BP3.Value;
IO_AI_T_BF1(
    ProcessError := ModbusWord_T_BF1.Error,
    ProcessValue := ModbusWord_T_BF1.Value,
    k := Parameters.Regulation.SupplyAir.KFactor); // FlowInput
IO_AI_F_BF1(
    ProcessError := ModbusWord_F_BF1.Error,
    ProcessValue := ModbusWord_F_BF1.Value,
    k := Parameters.Regulation.ExtractAir.KFactor); // FlowInput
IO_AI_T_BP1(ProcessError := ModbusWord_T_BP1.Error, ProcessValue := ModbusWord_T_BP1.Value); // PressureInput
IO_AI_F_BP1(ProcessError := ModbusWord_F_BP1.Error, ProcessValue := ModbusWord_F_BP1.Value); // PressureInput
IO_AI_T_BP2(
    ProcessError := ModbusWord_T_BP2.Error,
    ProcessValue := ModbusWord_T_BP2.Value,
    Override := T_BP2_Override,
    OverrideValue := T_BP2_OverrideValue); // PressureInput
IO_AI_F_BP2(ProcessError := ModbusWord_F_BP2.Error, ProcessValue := ModbusWord_F_BP2.Value); // PressureInput
IO_AI_F_BP3(ProcessError := ModbusWord_F_BP3.Error, ProcessValue := ModbusWord_F_BP3.Value); // PressureInput
Globals.IO.ModbusRTU.T_BP1 := ModbusWord_T_BP1.Value;
Globals.IO.ModbusRTU.T_BP1_Error := ModbusWord_T_BP1.Error;
Globals.IO.ModbusRTU.F_BP1 := ModbusWord_F_BP1.Value;
Globals.IO.ModbusRTU.F_BP1_Error := ModbusWord_F_BP1.Error;
Globals.IO.ModbusRTU.T_BP2 := ModbusWord_T_BP2.Value;
Globals.IO.ModbusRTU.T_BP2_Error := ModbusWord_T_BP2.Error;
Globals.IO.ModbusRTU.F_BP2 := ModbusWord_F_BP2.Value;
Globals.IO.ModbusRTU.F_BP2_Error := ModbusWord_F_BP2.Error;
Globals.IO.ModbusRTU.F_BP3 := ModbusWord_F_BP3.Value;
Globals.IO.ModbusRTU.F_BP3_Error := ModbusWord_F_BP3.Error;
Globals.IO.ModbusRTU.T_BF1_Error := ModbusWord_T_BF1.Error;
Globals.IO.ModbusRTU.F_BF1 := ModbusWord_F_BF1.Value;
Globals.IO.ModbusRTU.T_BF1 := ModbusWord_T_BF1.Value;
Globals.IO.ModbusRTU.F_BF1_Error := ModbusWord_F_BF1.Error;

// PAGE Fan power
EBM_Power_1(
    EN := EN and Parameters.Regulation.ExtractAir.FanType = FanTypes.EBM,
    ModbusRTU := ModbusRTU,
    Address := 102); // EBM_Power
F_CurrentPower := _w1;
T_CurrentPower := MUX(Parameters.Regulation.ExtractAir.FanType, EBM_Power_1.Power, Gebhardt_Power_1.Power);
EBM_Power_0(
    EN := EN and Parameters.Regulation.ExtractAir.FanType = FanTypes.EBM,
    ModbusRTU := ModbusRTU,
    Address := 101); // EBM_Power
_w1 := MUX(Parameters.Regulation.ExtractAir.FanType, EBM_Power_0.Power, Gebhardt_Power_0.Power);
Gebhardt_Power_0(
    EN := EN and Parameters.Regulation.ExtractAir.FanType = FanTypes.Gebhardt,
    ModbusRTU := ModbusRTU,
    Address := 101); // Gebhardt_Power
Gebhardt_Power_1(
    EN := EN and Parameters.Regulation.ExtractAir.FanType = FanTypes.Gebhardt,
    ModbusRTU := ModbusRTU,
    Address := 102); // Gebhardt_Power

// PAGE Fan speed
EBM_Speed_0(
    EN := EN and Parameters.Regulation.ExtractAir.FanType = FanTypes.EBM,
    ModbusRTU := ModbusRTU,
    Address := 101); // EBM_Speed
EBM_Speed_1(
    EN := EN and Parameters.Regulation.ExtractAir.FanType = FanTypes.EBM,
    ModbusRTU := ModbusRTU,
    Address := 102); // EBM_Speed
F_CurrentSpeed := MUX(Parameters.Regulation.ExtractAir.FanType, EBM_Speed_0.Speed, Gebhardt_Speed_0.Speed);
Gebhardt_Speed_0(
    EN := EN and Parameters.Regulation.ExtractAir.FanType = FanTypes.Gebhardt,
    ModbusRTU := ModbusRTU,
    Address := 101); // Gebhardt_Speed
T_CurrentSpeed := MUX(Parameters.Regulation.ExtractAir.FanType, EBM_Speed_1.Speed, Gebhardt_Speed_1.Speed);
Gebhardt_Speed_1(
    EN := EN and Parameters.Regulation.ExtractAir.FanType = FanTypes.Gebhardt,
    ModbusRTU := ModbusRTU,
    Address := 102); // Gebhardt_Speed

END_FUNCTION_BLOCK

// ---- DUTs/ModbusRTU/ModbusRTU.TcPOU
FUNCTION_BLOCK ModbusRTU EXTENDS Modbus
VAR_INPUT
	EN: BOOL;
END_VAR
VAR_OUTPUT
	ENO: BOOL;
END_VAR
VAR
	ModbusMaster: ModbusRtuMaster_KL6x22B;
	stMbErrId: ST_ModbusErrorDiagnostics;
	State: INT;
	aRegisterArray1: ARRAY [1..125] OF WORD;
	aRegisterCoil: ARRAY [1..250] OF BYTE;
	Param: REFERENCE TO ModbusIo;
	Delay: TON;
	StartFlag: BOOL;
	Counter: LINT;
END_VAR
VAR PERSISTENT
END_VAR

SUPER^();
ENO := EN;
Delay(IN := StartFlag, PT := T#250MS);
CASE State OF
	0:
		IF EN THEN	
			StartFlag := TRUE;	
			CurrentIoIndex := 0;
			IF IO[CurrentIoIndex] <> 0 AND Delay.Q THEN
				StartFlag := FALSE;
				State := 10;
			END_IF	
		END_IF
	10:
		Param REF= IO[CurrentIoIndex]^; 
		IF NOT Param.EN THEN
			State := 30;
		ELSE
			IF Param.RegisterType = ModbusRegisterType.Holdingregister THEN
				ModbusMaster.ReadRegs(
					UnitID := IO[CurrentIoIndex]^.UnitID, 
					Quantity := 1, 
					MBAddr := Param.Register, 
					cbLength := 2, 
					pMemoryAddr := ADR(aRegisterArray1), 
					Execute := TRUE, 
					Timeout := T#2S);
			ELSE			
				ModbusMaster.ReadInputRegs(
					UnitID := IO[CurrentIoIndex]^.UnitID, 
					Quantity := 1, 
					MBAddr := Param.Register, 
					cbLength := 2, 
					pMemoryAddr := ADR(aRegisterArray1), 
					Execute := TRUE, 
					Timeout := T#2S);
			END_IF
			IF  ModbusMaster.BUSY THEN
				State := 11;
			END_IF
		END_IF
	11:
		IF Param.RegisterType = ModbusRegisterType.Holdingregister THEN
			ModbusMaster.ReadRegs();
		ELSE
			ModbusMaster.ReadInputRegs();
		END_IF
		IF  ModbusMaster.Error or NOT ModbusMaster.BUSY THEN
			State := 20;
		END_IF
	20:
		IF Param.RegisterType = ModbusRegisterType.Holdingregister THEN
			ModbusMaster.ReadRegs();
		ELSE
			ModbusMaster.ReadInputRegs();
		END_IF
		IF ModbusMaster.Error THEN
			stMbErrId := ModbusMaster.ErrorDiagnostics;
			IF Param.RegisterType = ModbusRegisterType.Holdingregister THEN
				ModbusMaster.ReadRegs(Execute := FALSE);
			ELSE
				ModbusMaster.ReadInputRegs(Execute := FALSE);
			END_IF
			Param.IncErrorCount();
			Param.ErrorOUT := Param.GetErrorCount() > 5;
			ErrorCount := ErrorCount + 1;
			State := 30;
		ELSIF NOT ModbusMaster.BUSY THEN
			IF Param.RegisterType = ModbusRegisterType.Holdingregister THEN
				ModbusMaster.ReadRegs(Execute := FALSE);
			ELSE
				ModbusMaster.ReadInputRegs(Execute := FALSE);
			END_IF
			Param.ValueWord := aRegisterArray1[1];
			Param.ErrorOUT := FALSE;
			Param.ResetErrorCount();
			ReadCount := ReadCount + 1;
			State := 30;
		END_IF
	30:
		IF Param.RegisterType = ModbusRegisterType.Holdingregister THEN
			ModbusMaster.ReadRegs(Execute := FALSE);
		ELSE
			ModbusMaster.ReadInputRegs(Execute := FALSE);
		END_IF
		Counter := Counter + 1;
		CurrentIoIndex := CurrentIoIndex + 1;
		IF CurrentIoIndex >= IO_COUNT THEN
			CurrentIoIndex := 0;
		END_IF
		IF IO[CurrentIoIndex] <> 0 THEN
			State := 10;
		ELSE				
			State := 0;
		END_IF
END_CASE

END_FUNCTION_BLOCK

// ---- DUTs/ModbusRTU/ModbusReadWord.TcPOU
FUNCTION_BLOCK ModbusReadWord EXTENDS ModbusIo
VAR_INPUT
	Override: BOOL;
	OverrideValue: INT;
END_VAR
VAR_OUTPUT
	Value: INT;
	ValueW: WORD;
END_VAR
VAR
END_VAR
VAR PERSISTENT
END_VAR

SUPER^();
IF Override THEN
	Value := OverrideValue;
END_IF
ValueW := ValueWord;

PROPERTY ValueWord : WORD
GET
IF NOT Override THEN
	ValueWord := INT_TO_WORD(Value);
ELSE
	ValueWord := INT_TO_WORD(OverrideValue);
END_IF
END_GET
SET
IF NOT Override THEN
	Value := WORD_TO_INT(ValueWord);
ELSE
	Value := OverrideValue;
END_IF
END_SET
END_PROPERTY

END_FUNCTION_BLOCK

// ---- DUTs/IO/PressureInput.TcPOU
FUNCTION_BLOCK PressureInput EXTENDS AnalogInput
VAR_INPUT
	Range: LREAL := 32767;
END_VAR
VAR_OUTPUT
END_VAR
VAR
	Aver: Average;
END_VAR
VAR PERSISTENT
END_VAR

SUPER^();

METHOD FB_init : BOOL
VAR_INPUT
	bInitRetains : BOOL; // if TRUE, the retain variables are initialized (warm start / cold start)
	bInCopyCode : BOOL;  // if TRUE, the instance afterwards gets moved into the copy code (online change)
END_VAR
IF bInitRetains THEN
	ProcessMin := 0;
	ProcessMax := 30000;
	MinValue := 0;
	MaxValue := 30000;
END_IF
END_METHOD

METHOD GetValue : LREAL
VAR_INPUT
END_VAR
Aver(NewSample := (SUPER^.GetValue() / 32767) * Range);
GetValue := Aver.Value;
END_METHOD

END_FUNCTION_BLOCK

// ---- DUTs/IO/FlowInput.TcPOU
FUNCTION_BLOCK FlowInput EXTENDS AnalogInput
VAR_INPUT
	k: LREAL;
END_VAR
VAR_OUTPUT
END_VAR
VAR
	Aver: Average;
END_VAR
VAR PERSISTENT
END_VAR

SUPER^();

METHOD FB_init : BOOL
VAR_INPUT
	bInitRetains : BOOL; // if TRUE, the retain variables are initialized (warm start / cold start)
	bInCopyCode : BOOL;  // if TRUE, the instance afterwards gets moved into the copy code (online change)
END_VAR
IF bInitRetains THEN
	ProcessMin := 0;
	ProcessMax := 30000;
	MinValue := 0;
	MaxValue := 30000;
END_IF
END_METHOD

METHOD GetValue : LREAL
VAR_INPUT
END_VAR
VAR
	Pressure: LREAL;
END_VAR
Pressure := SUPER^.GetValue();
Aver(NewSample := PressureToFlow(Pressure, k));
GetValue := Aver.Value;
END_METHOD

END_FUNCTION_BLOCK

// ---- DUTs/Fans/PressureToFlow.TcPOU
FUNCTION PressureToFlow : LREAL
VAR_INPUT
	Pressure: LREAL;
	k: LREAL;
END_VAR
VAR
	DiffPressure: LREAL;
END_VAR

DiffPressure := Pressure;
IF diffpressure < 0 THEN
	DiffPressure := 0;
END_IF 
PressureToFlow := k * SQRT(DiffPressure);// / 3.6;

END_FUNCTION

// ---- DUTs/ModbusRTU/EBM_Power.TcPOU
FUNCTION_BLOCK EBM_Power
VAR_INPUT
	EN: BOOL;
	ModbusRTU: REFERENCE TO ModbusRTU;
	Address: BYTE := 101;
END_VAR
VAR_OUTPUT
	ENO: BOOL;
	Power: LREAL;
END_VAR
VAR
	ModbusWord_T_Power: ModbusReadWord;
	ModbusWord_T_RefU: ModbusReadWord;
	ModbusWord_T_RefI: ModbusReadWord;
	T_RefU: LREAL;
	T_RefI: LREAL;
END_VAR
VAR // added by the converter: edge detectors and wires of the graphical bodies
    _w1, _w2, _w4, _w5 : ANY;
    _w3 : LREAL;
END_VAR

ENO := EN;
Power := (_w1 * _w2) / 65536;
ModbusWord_T_Power(
    EN := EN,
    Modbus := ModbusRTU,
    UnitID := Address,
    RegisterType := ModbusRegisterType.InputRegister,
    Register := 16#d021); // ModbusReadWord
_w1 := WORD_TO_LREAL(ModbusWord_T_Power.ValueW);
_w3 := WORD_TO_LREAL(ModbusWord_T_RefU.ValueW);
ModbusWord_T_RefU(
    EN := EN,
    Modbus := ModbusRTU,
    UnitID := Address,
    RegisterType := ModbusRegisterType.HoldingRegister,
    Register := 16#d1a0); // ModbusReadWord
_w2 := _w4 * _w5;
_w4 := (_w3 * 20) / 1000;
T_RefU := _w4;
ModbusWord_T_RefI(
    EN := EN,
    Modbus := ModbusRTU,
    UnitID := Address,
    RegisterType := ModbusRegisterType.HoldingRegister,
    Register := 16#d1a1); // ModbusReadWord
_w5 := (WORD_TO_LREAL(ModbusWord_T_RefI.ValueW) * 2) / 1000;
T_RefI := _w5;

END_FUNCTION_BLOCK

// ---- DUTs/ModbusRTU/Gebhardt_Power.TcPOU
FUNCTION_BLOCK Gebhardt_Power
VAR_INPUT
	EN: BOOL;
	ModbusRTU: REFERENCE TO ModbusRTU;
	Address: BYTE := 101;
END_VAR
VAR_OUTPUT
	ENO: BOOL;
	Power: LREAL;
END_VAR
VAR
	ModbusWord_T_Power: ModbusReadWord;
END_VAR
VAR // added by the converter: edge detectors and wires of the graphical bodies
    _w1 : LREAL;
END_VAR

ENO := EN;
Power := _w1;
ModbusWord_T_Power(
    EN := EN,
    Modbus := ModbusRTU,
    UnitID := Address,
    RegisterType := ModbusRegisterType.InputRegister,
    Register := 31); // ModbusReadWord
_w1 := WORD_TO_LREAL(ModbusWord_T_Power.ValueW);

END_FUNCTION_BLOCK

// ---- DUTs/ModbusRTU/EBM_Speed.TcPOU
FUNCTION_BLOCK EBM_Speed
VAR_INPUT
	EN: BOOL;
	ModbusRTU: REFERENCE TO ModbusRTU;
	Address: BYTE := 101;
END_VAR
VAR_OUTPUT
	ENO: BOOL;
	Speed: LREAL;
END_VAR
VAR
	ModbusWord_T_ActualSpeed: ModbusReadWord;
	ModbusWord_T_nMax: ModbusReadWord;
	ActualSpeed: LREAL;
END_VAR
VAR // added by the converter: edge detectors and wires of the graphical bodies
    _w1 : ANY;
    _w2 : LREAL;
END_VAR

ENO := EN;
_w2 := (_w1 * TO_LREAL(ModbusWord_T_nMax.ValueW)) / 64000;
ModbusWord_T_ActualSpeed(
    EN := EN,
    Modbus := ModbusRTU,
    UnitID := Address,
    RegisterType := ModbusRegisterType.InputRegister,
    Register := 16#d010); // ModbusReadWord
_w1 := TO_LREAL(ModbusWord_T_ActualSpeed.ValueW);
Speed := _w2;
ModbusWord_T_nMax(
    EN := EN,
    Modbus := ModbusRTU,
    UnitID := Address,
    RegisterType := ModbusRegisterType.HoldingRegister,
    Register := 16#d119); // ModbusReadWord

END_FUNCTION_BLOCK

// ---- DUTs/ModbusRTU/Gebhardt_Speed.TcPOU
FUNCTION_BLOCK Gebhardt_Speed
VAR_INPUT
	EN: BOOL;
	ModbusRTU: REFERENCE TO ModbusRTU;
	Address: BYTE := 101;
END_VAR
VAR_OUTPUT
	ENO: BOOL;
	Speed: LREAL;
END_VAR
VAR
	ModbusWord_T_Speed: ModbusReadWord;
END_VAR

ENO := EN;
Speed := WORD_TO_LREAL(ModbusWord_T_Speed.ValueW);
ModbusWord_T_Speed(
    EN := EN,
    Modbus := ModbusRTU,
    UnitID := Address,
    RegisterType := ModbusRegisterType.InputRegister,
    Register := 31); // ModbusReadWord

END_FUNCTION_BLOCK

// ---- POUs/TestPID.TcPOU
FUNCTION_BLOCK TestPID
VAR_INPUT
END_VAR
VAR_OUTPUT
END_VAR
VAR
	Ramp: Ramp;
	PidController: PidController;
	Target: lreal := 1;
END_VAR

PidController(SP := 100, PV := 90, SyncCV := Ramp.Value, Sync := Ramp.Value < 0.75);
Ramp(Target := Target);

END_FUNCTION_BLOCK

// ---- POUs/Timers.TcPOU
PROGRAM Timers
VAR
	SecondsTimer: Timer;
	LastTime, Now: LINT;
	InitDone: BOOL;
	BlinkPeriod: INT;
	CurrentBlinkPeriod: INT;
END_VAR

IF NOT InitDone THEN
	Now := SecondsTimer.ElapsedTime();
	InitDone := TRUE;
END_IF

// Show that we are alive
Globals.LifeCounter := Globals.LifeCounter + 1;

// Count seconds
Globals.SecondsCounter := SecondsTimer.ElapsedTime() / 1000;

IF Main.GreenMaster.VentilationRunning THEN
	IF Main.GreenMaster.TemperatureControlRunning THEN
		BlinkPeriod := 250;
	ELSE
		BlinkPeriod := 1000;
	END_IF
ELSE
	BlinkPeriod := 3000;
END_IF

IF BlinkPeriod <> CurrentBlinkPeriod THEN
	LastTime := SecondsTimer.ElapsedTime();
END_IF

IF Main.GreenMaster.Parameters.System.Operation.EN THEN
	// Blink ERR LED
	Now := SecondsTimer.ElapsedTime();
	IF (Now - LastTime) > (BlinkPeriod - 50) THEN
		F_CX8190_LED_ERR(eMode := E_CX81x0_LED.eCX81x0_LED_GREEN_ON);
	END_IF
	IF (Now - LastTime) > BlinkPeriod THEN
		F_CX8190_LED_ERR(eMode := E_CX81x0_LED.eCX81x0_LED_GREEN_OFF);
		LastTime := LastTime + BlinkPeriod; 
	END_IF
ELSE
	F_CX8190_LED_ERR(eMode := E_CX81x0_LED.eCX81x0_LED_RED_ON);
END_IF
CurrentBlinkPeriod := BlinkPeriod;

END_PROGRAM

// ---- DUTs/Alarms/AlarmHandler.TcPOU
FUNCTION_BLOCK AlarmHandler
VAR_INPUT
END_VAR
VAR_OUTPUT
END_VAR
VAR
END_VAR

// Check for alarms

METHOD GetAlarm : reference to AlarmDef
VAR_INPUT
	{attribute 'TcEncoding':='UTF-8'}
	Name: string;
END_VAR
VAR
	n: INT;
END_VAR
GetAlarm REF= 0;
FOR n := 0 TO GlobalSettings.MAX_ALARMS - 1 DO
	IF GlobalSettings.AlarmDefs[n].Name = '' THEN
		EXIT;
	END_IF
	IF GlobalSettings.AlarmDefs[n].Name = Name THEN
		GetAlarm REF= GlobalSettings.AlarmDefs[n];
		EXIT;
	END_IF
END_FOR
END_METHOD

END_FUNCTION_BLOCK

// ---- DUTs/Custom/ParallelUnits/ParallelUnits.TcPOU
FUNCTION_BLOCK ParallelUnits
VAR_INPUT
	EN: BOOL;
	Tags: REFERENCE TO AdsTagsParallelUnits;
	Parameters: REFERENCE TO GreenMasterBaseParameters;
END_VAR
VAR_OUTPUT
	FireSupplyAlarm: BOOL;
	FireExtractAlarm: BOOL;
	FreezeAlarm: bool;
	RemoteStatusData: RemoteStatusData;
END_VAR
VAR
	LocalAmsNumber: LINT;
	RemoteAmsNumber: LINT;
	RemoteOrderToSend: RemoteOrder;
	Week: WORD;
	FirstTime: BOOL;
	HostName: FB_GetHostName;
	FoundHost: BOOL;
	StateTime: Timer;
	RemoteActive: BOOL;
	InstantaneousDualNeeded: BOOL;
	DualNeeded: BOOL;
	DualNeededTON: TON;
	DualNeededTOF: TOF;
	Runnable: BOOL;
	CanBeRunnable: BOOL;
	RemoteValidTOF: TOF;
	AddWeekTest: WORD;
	TransferOk: BOOL;
	TransferTON: TON;
	TempSP: LREAL;
	SupplyAirSetPointAdjustmentFB: SetPointAdjustmentFB;
	ExtractAirSetPointAdjustmentFB: SetPointAdjustmentFB;
	SupplyAirSetPointAdjustmentFB_HighSpeed: SetPointAdjustmentFB;
	ExtractAirSetPointAdjustmentFB_HighSpeed: SetPointAdjustmentFB;
	StandaloneSupplyAirSetPointAdjustmentFB: SetPointAdjustmentFB;
	StandaloneExtractAirSetPointAdjustmentFB: SetPointAdjustmentFB;
	StandaloneSupplyAirSetPointAdjustmentFB_HighSpeed: SetPointAdjustmentFB;
	StandaloneExtractAirSetPointAdjustmentFB_HighSpeed: SetPointAdjustmentFB;
	SupplyAirPressureDeviation: DeviationMonitor;
	ExtractAirPressureDeviation: DeviationMonitor;
	CurrentFireSupply: BOOL;
	CurrentFireExtract: BOOL;
	IsAlarm: BOOL;
	LastResetAlarmsCounter: INT;
	ResetAlarmsTOF: TOF;
END_VAR

IF NOT FirstTime THEN
	HostName(bExecute := TRUE);
	IF NOT HostName.bBusy THEN	
		FoundHost := FALSE;
		// E6
		IF F_ToUCase(HostName.sHostName) = 'STU_E6-LB01' THEN
			Tags.Settings.RemoteAmsId := '10.138.21.151.1.1';
			Tags.Status.isMaster := TRUE;
			FoundHost := TRUE;
		ELSIF F_ToUCase(HostName.sHostName) = 'STU_E6-LB02' THEN
			Tags.Settings.RemoteAmsId := '10.138.21.150.1.1';
			Tags.Status.isMaster := FALSE;
			FoundHost := TRUE;
		END_IF
		// E1
		IF F_ToUCase(HostName.sHostName) = 'STU_E1-LB01' THEN
			Tags.Settings.RemoteAmsId := '10.138.21.153.1.1';
			Tags.Status.isMaster := TRUE;
			FoundHost := TRUE;
		ELSIF F_ToUCase(HostName.sHostName) = 'STU_E1-LB02' THEN
			Tags.Settings.RemoteAmsId := '10.138.21.152.1.1';
			Tags.Status.isMaster := FALSE;
			FoundHost := TRUE;
		END_IF
		// DIGINET Test system
		IF F_ToUCase(HostName.sHostName) = 'DIGINET-1' THEN
			Tags.Settings.RemoteAmsId := '5.102.41.153.1.1';
			Tags.Status.isMaster := TRUE;
			FoundHost := TRUE;
		ELSIF F_ToUCase(HostName.sHostName) = 'DIGINET-2' THEN
			Tags.Settings.RemoteAmsId := '5.73.47.143.1.1';
			Tags.Status.isMaster := FALSE;
			FoundHost := TRUE;
		END_IF
		// NIBE AirSite Test system
		IF F_ToUCase(HostName.sHostName) = 'AIRPLC-DEMO' THEN
			Tags.Settings.RemoteAmsId := '5.102.42.161.1.1';
			Tags.Status.isMaster := TRUE;
			FoundHost := TRUE;
		ELSIF F_ToUCase(HostName.sHostName) = 'CX-662AA1' THEN
			Tags.Settings.RemoteAmsId := '10.133.0.22.1.1';
			Tags.Status.isMaster := FALSE;
			FoundHost := TRUE;
		END_IF
		IF NOT FoundHost THEN
			Tags.Status.isMaster := TRUE;			
		END_IF
		Tags.Status.isSlave := NOT Tags.Status.isMaster;
		// First time or remote AMS ID changed
		FirstTime := TRUE;
	END_IF
END_IF
StateTime();
Runnable := Parameters.System.Operation.State = SystemStates.Run;
CanBeRunnable := Main.GreenMaster.Runnable(IncludeSP := FALSE);
Tags.Status.CanBeRunnable := CanBeRunnable;
IF Runnable THEN
	IF NOT InstantaneousDualNeeded THEN
		IF (Parameters.Regulation.SupplyAir.Control.CV > Tags.Settings.StandaloneMaxFan) OR
			(Parameters.Regulation.ExtractAir.Control.CV > Tags.Settings.StandaloneMaxFan) OR
			(RemoteStatusData.RemoteStatus.SupplyFanSpeed > Tags.Settings.StandaloneMaxFan) OR
			(RemoteStatusData.RemoteStatus.ExtractFanSpeed > Tags.Settings.StandaloneMaxFan) THEN
			InstantaneousDualNeeded := TRUE;
		END_IF
	ELSE
		IF (Parameters.Regulation.SupplyAir.Control.CV < Tags.Settings.DualMinFan) AND
			(Parameters.Regulation.ExtractAir.Control.CV < Tags.Settings.DualMinFan) AND
			(RemoteStatusData.RemoteStatus.SupplyFanSpeed < Tags.Settings.DualMinFan) AND
			(RemoteStatusData.RemoteStatus.ExtractFanSpeed < Tags.Settings.DualMinFan) THEN
			InstantaneousDualNeeded := FALSE;
		END_IF
	END_IF
	DualNeededTON(IN := InstantaneousDualNeeded, PT := T#5M);
	DualNeededTOF(IN := InstantaneousDualNeeded, PT := T#5M);
	IF NOT DualNeeded THEN
		IF DualNeededTON.Q THEN
			DualNeeded := TRUE;
		END_IF
	ELSE
		IF NOT DualNeededTOF.Q THEN
			DualNeeded := FALSE;
		END_IF
	END_IF
END_IF
Week := F_GetWeekOfTheYear(NowDT()) + AddWeekTest;;
RemoteValidTOF(IN := RemoteStatusData.Valid, PT := T#10S); 
RemoteActive := RemoteValidTOF.Q AND RemoteStatusData.RemoteStatus.IsRunning;
Tags.Status.SupplyFanSpeed := Parameters.Regulation.SupplyAir.Control.CV;
Tags.Status.ExtractFanSpeed := Parameters.Regulation.ExtractAir.Control.CV;
Tags.Status.IsRunning := Parameters.IO.DIn.Auto;
Tags.Status.State := Parameters.System.Operation.State;
ResetAlarmsTOF(IN := Globals.ResetAlarmsCounter <> LastResetAlarmsCounter, PT := T#2S);
LastResetAlarmsCounter := Globals.ResetAlarmsCounter;
IF Tags.Status.IsMaster THEN
	Tags.Status.ResetAlarmMaster := ResetAlarmsTOF.Q;
ELSE
	Tags.Status.ResetAlarmSlave := ResetAlarmsTOF.Q;
END_IF

CurrentFireSupply := Parameters.IO.DIn.FireSupplyAlarm;
CurrentFireExtract := Parameters.IO.DIn.FireExtractAlarm OR 
	Parameters.Alarm.Status.A.FireExtractExternal OR 
	Parameters.Alarm.Status.A.FireExtractPressure OR 
	Parameters.Alarm.Status.A.FireExtractTemperature;
IF Tags.Status.IsMaster THEN
	Tags.Status.FireSupplyMaster := CurrentFireSupply;
	Tags.Status.FireExtractMaster := CurrentFireExtract;
	Tags.Status.FreezeMaster := Main.CurrentFreezeAlarm;
ELSE
	Tags.Status.FireSupplySlave := CurrentFireSupply;
	Tags.Status.FireExtractSlave := CurrentFireExtract;
	Tags.Status.FreezeSlave := Main.CurrentFreezeAlarm;
END_IF
Tags.Status.PressureSupplyCSP := GetSetPointSupply();
Tags.Status.PressureExtractCSP := GetSetPointExtract();
CurrentFireSupply := Parameters.Alarm.Active.A.FireExtract OR 
						Parameters.Alarm.Active.A.FireExtractExternal OR 
						Parameters.Alarm.Active.A.FireExtractPressure OR 
						Parameters.Alarm.Active.A.FireExtractTemperature OR 
						Parameters.Alarm.Active.A.FireLocal OR
						Parameters.Alarm.Active.A.FireSupply;
IsAlarm := CurrentFireSupply OR Parameters.Alarm.Active.A.Freeze;

// Check pressure deviation
SupplyAirPressureDeviation(	EN := Tags.Status.IsMaster AND (Parameters.System.Operation.State = SystemStates.Run),
							TargetValue := GetSetPointSupply(),
							DiffAllowed := Parameters.Alarm.Limits.B.SupplyAirPressureDeviation,
							Mode := DeviationMonitorMode.Diff,
							Value := Parameters.IO.AIn.F_BP1,
							OnDelay := LTIME#0S
);
IF Parameters.Regulation.SupplyAir.ControlMode = FanControlTypes.Const THEN
	Parameters.Alarm.Status.B.SupplyAirDeviation := SupplyAirPressureDeviation.Error;	
END_IF

ExtractAirPressureDeviation(	EN := Tags.Status.IsMaster AND (Parameters.System.Operation.State = SystemStates.Run),
							TargetValue := GetSetPointExtract(),
							DiffAllowed := Parameters.Alarm.Limits.B.ExtractAirPressureDeviation,
							Mode := DeviationMonitorMode.Diff,
							Value := Parameters.IO.AIn.T_BP1,
							OnDelay := LTIME#0S
);
IF Parameters.Regulation.ExtractAir.ControlMode = FanControlTypes.Const THEN
	Parameters.Alarm.Status.B.ExtractAirDeviation := ExtractAirPressureDeviation.Error;	
END_IF

IF FirstTime THEN
	MasterSlave();
END_IF
IF EN THEN
	TransferTON(IN := TRUE, PT := T#300ms);
	IF TransferTON.Q THEN
		TransferTON(IN := FALSE);
		RemoteStatusData := ReadFromRemote();
		IF RemoteStatusData.Valid THEN
			IF Tags.Status.IsMaster THEN
				Parameters.Alarm.Control.ResetAlarms := RemoteStatusData.RemoteStatus.ResetAlarmSlave;
			ELSE
				Parameters.Alarm.Control.ResetAlarms := RemoteStatusData.RemoteStatus.ResetAlarmMaster;
			END_IF
			IF Tags.Status.IsMaster THEN
				FireSupplyAlarm := RemoteStatusData.RemoteStatus.FireSupplySlave;
				FireExtractAlarm := RemoteStatusData.RemoteStatus.FireExtractSlave;
				FreezeAlarm := RemoteStatusData.RemoteStatus.FreezeSlave;
			ELSE
				FireSupplyAlarm := RemoteStatusData.RemoteStatus.FireSupplyMaster;
				FireExtractAlarm := RemoteStatusData.RemoteStatus.FireExtractMaster;
				FreezeAlarm := RemoteStatusData.RemoteStatus.FreezeMaster;
			END_IF
			RemoteOrderToSend.Counter := RemoteOrderToSend.Counter + 1;
			IF Tags.Status.IsMaster THEN
				RemoteOrderToSend.TimeChannels := Parameters.System.Operation.TimeChannels;
				RemoteOrderToSend.TemperatureControl := Parameters.Regulation.Temperature.Control;		
				RemoteOrderToSend.TemperatureSetPointAdjustment := Parameters.Regulation.Temperature.SetPointAdjustment;
				RemoteOrderToSend.SupplyAirSetPointAdjustment := Tags.Settings.SupplyAirSetPointAdjustment;
				RemoteOrderToSend.ExtractAirSetPointAdjustment := Tags.Settings.ExtractAirSetPointAdjustment;
				RemoteOrderToSend.NightCoolingRequest := Parameters.Regulation.NightCoolingRequest;
				RemoteOrderToSend.DualExtractSP := Tags.Settings.PressureExtractSP; 
				RemoteOrderToSend.DualExtractSP_HighSpeed := Tags.Settings.PressureExtractSP_HighSpeed; 
				RemoteOrderToSend.DualSupplySP := Tags.Settings.PressureSupplySP; 
				RemoteOrderToSend.DualSupplySP_HighSpeed := Tags.Settings.PressureSupplySP_HighSpeed; 
			END_IF
			TransferOk := TransferToRemote(sNetId := Tags.Settings.RemoteAmsId, Src := RemoteOrderToSend, Dest := 'ADS_ParallelUnits.Tags.Settings.RemoteOrder');	
			IF RemoteValidTOF.Q AND Tags.Status.IsSlave AND (Tags.Settings.RemoteOrder.Counter <> 0) THEN
				Parameters.System.Operation.TimeChannels := Tags.Settings.RemoteOrder.TimeChannels;	
				Parameters.Regulation.Temperature.Control.SP := Tags.Settings.RemoteOrder.TemperatureControl.SP;		
				Parameters.Regulation.Temperature.Control.SP_HighSpeed := Tags.Settings.RemoteOrder.TemperatureControl.SP;		
				Parameters.Regulation.Temperature.SetPointAdjustment := Tags.Settings.RemoteOrder.TemperatureSetPointAdjustment;		
				Tags.Settings.SupplyAirSetPointAdjustment := Tags.Settings.RemoteOrder.SupplyAirSetPointAdjustment;		
				Tags.Settings.ExtractAirSetPointAdjustment := Tags.Settings.RemoteOrder.ExtractAirSetPointAdjustment;	
				Parameters.Regulation.NightCoolingRequest := Tags.Settings.RemoteOrder.NightCoolingRequest;
				Tags.Settings.PressureExtractSP := TO_REAL(Tags.Settings.RemoteOrder.DualExtractSP);
				Tags.Settings.PressureExtractSP_HighSpeed := TO_REAL(Tags.Settings.RemoteOrder.DualExtractSP_HighSpeed);
				Tags.Settings.PressureSupplySP := TO_REAL(Tags.Settings.RemoteOrder.DualSupplySP);
				Tags.Settings.PressureSupplySP_HighSpeed := TO_REAL(Tags.Settings.RemoteOrder.DualSupplySP_HighSpeed);
			END_IF
		ELSE
			IF Tags.Status.IsSlave THEN
				Parameters.Regulation.NightCoolingRequest := FALSE;
			END_IF
			FireSupplyAlarm := FALSE;
			FreezeAlarm := FALSE;
		END_IF		
	END_IF
END_IF

METHOD GetAmsNumbers : BOOL
VAR_INPUT
END_VAR
VAR_INST
	LocalAddrBytes: AMSNETID;
	RemoteAddrBytes: AMSNETID;	
	FB_GetLocalAmsNetId: FB_GetLocalAmsNetId;
	UsedRemoteAmsId: string := '???';
END_VAR
IF Tags.Settings.RemoteAmsId <> UsedRemoteAmsId THEN
	UsedRemoteAmsId := Tags.Settings.RemoteAmsId;
	RemoteAddrBytes := F_ScanAmsNetIds(Tags.Settings.RemoteAmsId);
	FB_GetLocalAmsNetId(bExecute := TRUE, AddrBytes => LocalAddrBytes);
	FB_GetLocalAmsNetId(bExecute := FALSE);
	IF NOT FB_GetLocalAmsNetId.bBusy AND NOT FB_GetLocalAmsNetId.bError THEN			
		LocalAmsNumber := 	
						SHL(TO_LINT(LocalAddrBytes[0]),  40) + 
						SHL(TO_LINT(LocalAddrBytes[1]),  32) + 
						SHL(TO_LINT(LocalAddrBytes[2]),  24) + 
						SHL(TO_LINT(LocalAddrBytes[3]), 16) + 
						SHL(TO_LINT(LocalAddrBytes[4]), 8) + 
						TO_LINT(LocalAddrBytes[5]); 
		RemoteAmsNumber := 	
						SHL(TO_LINT(RemoteAddrBytes[0]),  40) + 
						SHL(TO_LINT(RemoteAddrBytes[1]),  32) + 
						SHL(TO_LINT(RemoteAddrBytes[2]),  24) + 
						SHL(TO_LINT(RemoteAddrBytes[3]), 16) + 
						SHL(TO_LINT(RemoteAddrBytes[4]), 8) + 
						TO_LINT(RemoteAddrBytes[5]); 
	END_IF
	GetAmsNumbers := TRUE;
ELSE 
	GetAmsNumbers := FALSE;
END_IF
END_METHOD

METHOD GetSetPointExtract : REAL
VAR_INPUT
END_VAR
VAR
	TempSP: REAL;
END_VAR
IF Parameters.Regulation.NightCooling OR 
	Parameters.IO.DIn.ExtendedOperation OR 
	Parameters.System.Operation.TimeChannels.HighSpeed OR 
	(ADS_Standard.Tags.Settings.RemoteStart = 2) THEN
	TempSP := Tags.Settings.PressureExtractSP_HighSpeed;
	ExtractAirSetPointAdjustmentFB_HighSpeed(X := Parameters.Regulation.CompensationTemperature, SetPointAdjustment := Tags.Settings.ExtractAirSetPointAdjustment);
	GetSetPointExtract := TO_REAL(Tags.Settings.ExtractAirSetPointAdjustment.Y) + TempSP;
ELSE
	TempSP := Tags.Settings.PressureExtractSP;
	ExtractAirSetPointAdjustmentFB(X := Parameters.Regulation.CompensationTemperature, SetPointAdjustment := Tags.Settings.ExtractAirSetPointAdjustment);
	GetSetPointExtract := TO_REAL(Tags.Settings.ExtractAirSetPointAdjustment.Y) + TempSP;
END_IF
END_METHOD

METHOD GetSetPointSupply : REAL
VAR_INPUT
END_VAR
VAR
	TempSP: REAL;
END_VAR
IF Parameters.Regulation.NightCooling OR 
	Parameters.IO.DIn.ExtendedOperation OR 
	Parameters.System.Operation.TimeChannels.HighSpeed OR 
	(ADS_Standard.Tags.Settings.RemoteStart = 2) THEN
	TempSP := Tags.Settings.PressureSupplySP_HighSpeed;
	SupplyAirSetPointAdjustmentFB_HighSpeed(X := Parameters.Regulation.CompensationTemperature, SetPointAdjustment := Tags.Settings.SupplyAirSetPointAdjustment);
	GetSetPointSupply := TO_REAL(Tags.Settings.SupplyAirSetPointAdjustment.Y) + TempSP;
ELSE
	TempSP := Tags.Settings.PressureSupplySP;
	SupplyAirSetPointAdjustmentFB(X := Parameters.Regulation.CompensationTemperature, SetPointAdjustment := Tags.Settings.SupplyAirSetPointAdjustment);
	GetSetPointSupply := TO_REAL(Tags.Settings.SupplyAirSetPointAdjustment.Y) + TempSP;
END_IF
END_METHOD

METHOD MasterCanRun : BOOL
VAR_INPUT
END_VAR
MasterCanRun := CanBeRunnable;
END_METHOD

METHOD MasterSlave : BOOL
VAR_INPUT
END_VAR
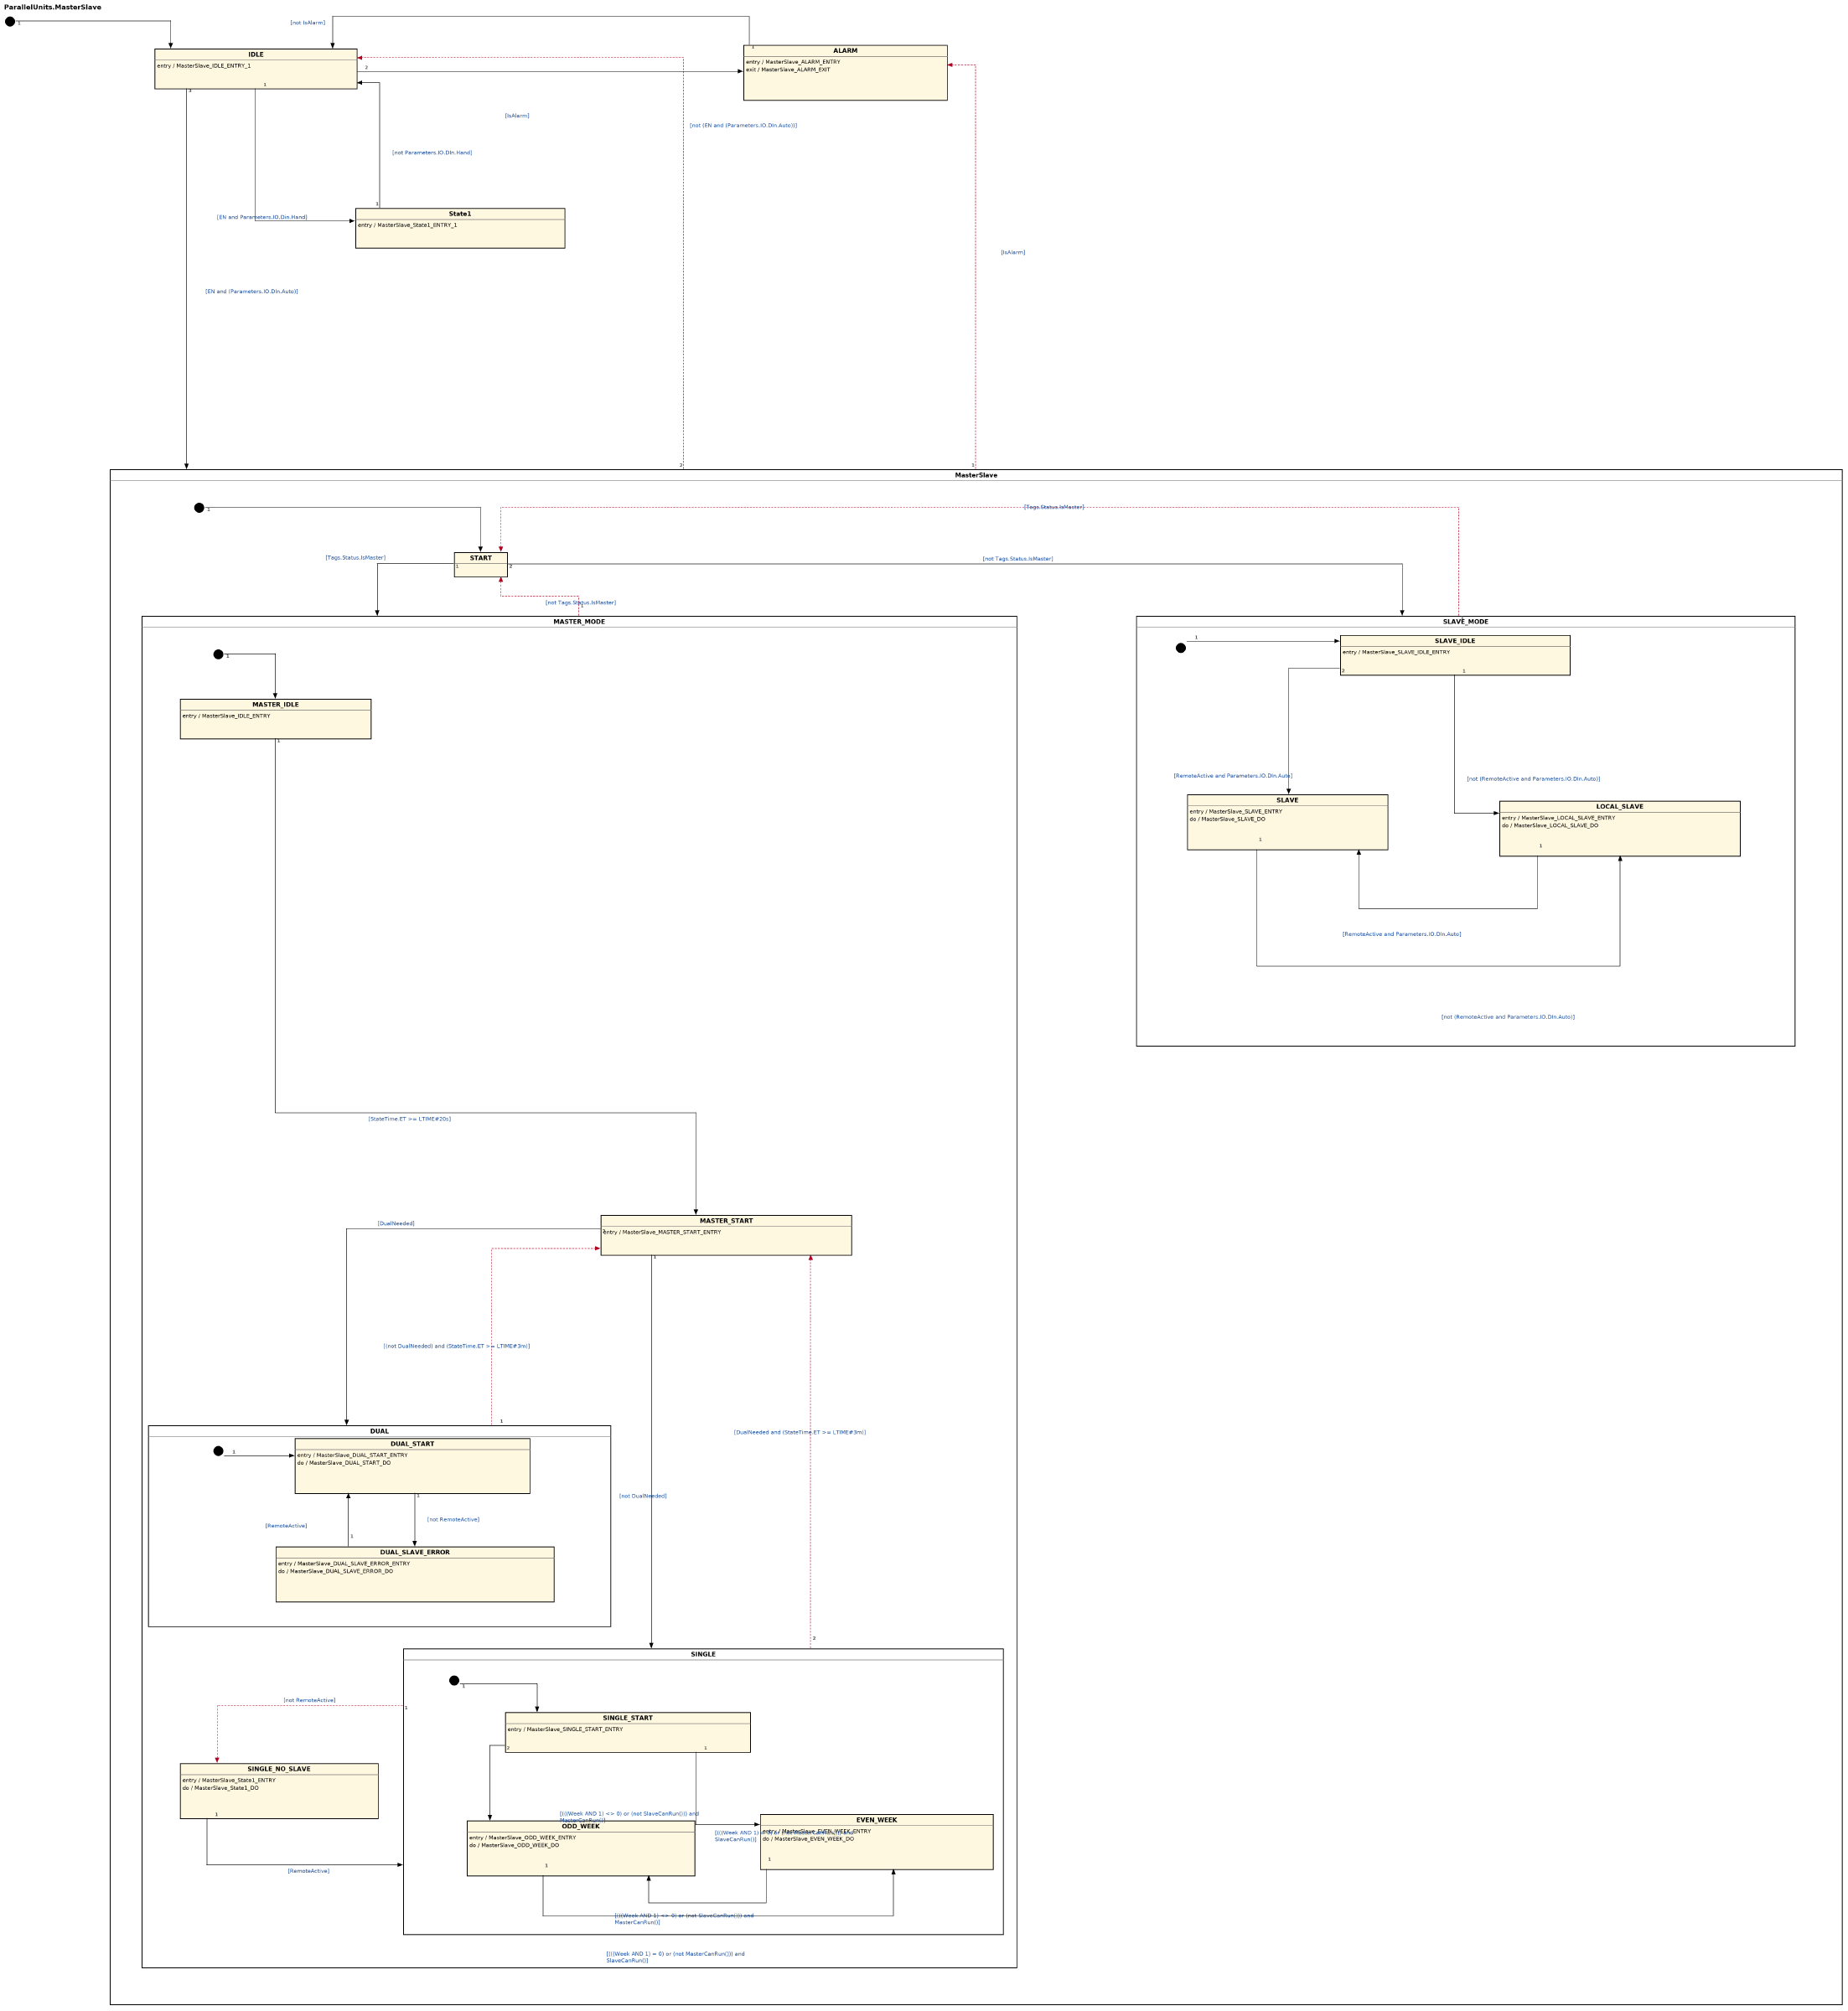
STATECHART MasterSlave  // abortable
    START StartState2
    STATE ALARM
        entry / MasterSlave_ALARM_ENTRY
        exit / MasterSlave_ALARM_EXIT
    STATE IDLE
        entry / MasterSlave_IDLE_ENTRY_1
    STATE State1
        entry / MasterSlave_State1_ENTRY_1
    COMPOSITE STATE MasterSlave
        START StartState1
        STATE START
        COMPOSITE STATE MASTER_MODE
            START StartState6
            STATE MASTER_IDLE
                entry / MasterSlave_IDLE_ENTRY
            STATE MASTER_START
                entry / MasterSlave_MASTER_START_ENTRY
            COMPOSITE STATE DUAL
                START StartState4
                STATE DUAL_START
                    entry / MasterSlave_DUAL_START_ENTRY
                    do / MasterSlave_DUAL_START_DO
                STATE DUAL_SLAVE_ERROR
                    entry / MasterSlave_DUAL_SLAVE_ERROR_ENTRY
                    do / MasterSlave_DUAL_SLAVE_ERROR_DO
                StartState4 -> DUAL_START  // priority 1, on completion
                DUAL_START -> DUAL_SLAVE_ERROR [not RemoteActive] // priority 1
                DUAL_SLAVE_ERROR -> DUAL_START [RemoteActive] // priority 1
            END_STATE
            COMPOSITE STATE SINGLE
                START StartState3
                STATE SINGLE_START
                    entry / MasterSlave_SINGLE_START_ENTRY
                STATE ODD_WEEK
                    entry / MasterSlave_ODD_WEEK_ENTRY
                    do / MasterSlave_ODD_WEEK_DO
                STATE EVEN_WEEK
                    entry / MasterSlave_EVEN_WEEK_ENTRY
                    do / MasterSlave_EVEN_WEEK_DO
                StartState3 -> SINGLE_START  // priority 1, on completion
                SINGLE_START -> EVEN_WEEK [(((Week AND 1) = 0) or (not MasterCanRun())) and SlaveCanRun()] // priority 1
                SINGLE_START -> ODD_WEEK [(((Week AND 1) <> 0) or (not SlaveCanRun())) and MasterCanRun()] // priority 2
                ODD_WEEK -> EVEN_WEEK [(((Week AND 1) = 0) or (not MasterCanRun())) and SlaveCanRun()] // priority 1
                EVEN_WEEK -> ODD_WEEK [(((Week AND 1) <> 0) or (not SlaveCanRun())) and MasterCanRun()] // priority 1
            END_STATE
            STATE SINGLE_NO_SLAVE
                entry / MasterSlave_State1_ENTRY
                do / MasterSlave_State1_DO
            StartState6 -> MASTER_IDLE  // priority 1, on completion
            MASTER_IDLE -> MASTER_START [StateTime.ET >= LTIME#20s] // priority 1
            MASTER_START -> SINGLE [not DualNeeded] // priority 1
            MASTER_START -> DUAL [DualNeeded] // priority 2
            DUAL -> MASTER_START [(not DualNeeded) and (StateTime.ET >= LTIME#3m)] // priority 1, exception
            SINGLE -> SINGLE_NO_SLAVE [not RemoteActive] // priority 1, exception
            SINGLE -> MASTER_START [DualNeeded and (StateTime.ET >= LTIME#3m)] // priority 2, exception
            SINGLE_NO_SLAVE -> SINGLE [RemoteActive] // priority 1
        END_STATE
        COMPOSITE STATE SLAVE_MODE
            START StartState5
            STATE SLAVE_IDLE
                entry / MasterSlave_SLAVE_IDLE_ENTRY
            STATE SLAVE
                entry / MasterSlave_SLAVE_ENTRY
                do / MasterSlave_SLAVE_DO
            STATE LOCAL_SLAVE
                entry / MasterSlave_LOCAL_SLAVE_ENTRY
                do / MasterSlave_LOCAL_SLAVE_DO
            StartState5 -> SLAVE_IDLE  // priority 1, on completion
            SLAVE_IDLE -> LOCAL_SLAVE [not (RemoteActive and Parameters.IO.DIn.Auto)] // priority 1
            SLAVE_IDLE -> SLAVE [RemoteActive and Parameters.IO.DIn.Auto] // priority 2
            SLAVE -> LOCAL_SLAVE [not (RemoteActive and Parameters.IO.DIn.Auto)] // priority 1
            LOCAL_SLAVE -> SLAVE [RemoteActive and Parameters.IO.DIn.Auto] // priority 1
        END_STATE
        StartState1 -> START  // priority 1, on completion
        START -> MASTER_MODE [Tags.Status.IsMaster] // priority 1
        START -> SLAVE_MODE [not Tags.Status.IsMaster] // priority 2
        MASTER_MODE -> START [not Tags.Status.IsMaster] // priority 1, exception
        SLAVE_MODE -> START [Tags.Status.IsMaster] // priority 1, exception
    END_STATE
    StartState2 -> IDLE  // priority 1, on completion
    ALARM -> IDLE [not IsAlarm] // priority 1
    IDLE -> State1 [EN and Parameters.IO.Din.Hand] // priority 1
    IDLE -> ALARM [IsAlarm] // priority 2
    IDLE -> MasterSlave [EN and (Parameters.IO.DIn.Auto)] // priority 3
    State1 -> IDLE [not Parameters.IO.DIn.Hand] // priority 1
    MasterSlave -> ALARM [IsAlarm] // priority 1, exception
    MasterSlave -> IDLE [not (EN and (Parameters.IO.DIn.Auto))] // priority 2, exception
END_STATECHART
END_METHOD

METHOD MasterSlave_ALARM_ENTRY : BOOL
VAR_INPUT
END_VAR
Parameters.System.Operation.EN := FALSE;
END_METHOD

METHOD MasterSlave_ALARM_EXIT : BOOL
VAR_INPUT
END_VAR
Parameters.System.Operation.EN := TRUE;
END_METHOD

METHOD MasterSlave_DUAL_SLAVE_ERROR_DO : BOOL
VAR_INPUT
END_VAR
Parameters.Regulation.SupplyAir.Control.SP := GetSetPointSupply();
Parameters.Regulation.ExtractAir.Control.SP := GetSetPointExtract();
Parameters.Regulation.SupplyAir.Control.SP_HighSpeed := Parameters.Regulation.SupplyAir.Control.SP;
Parameters.Regulation.ExtractAir.Control.SP_HighSpeed := Parameters.Regulation.ExtractAir.Control.SP;
END_METHOD

METHOD MasterSlave_DUAL_SLAVE_ERROR_ENTRY : BOOL
VAR_INPUT
END_VAR
Parameters.Regulation.SupplyAir.ControlMode := FanControlTypes.Pressure;
Parameters.Regulation.ExtractAir.ControlMode := FanControlTypes.Pressure;
END_METHOD

METHOD MasterSlave_DUAL_START_DO : BOOL
VAR_INPUT
END_VAR
Parameters.Regulation.SupplyAir.Control.SP := PidControlSupplyAir(Sync := FALSE, SyncCV := 0);
Parameters.Regulation.ExtractAir.Control.SP := PidControlExtractAir(Sync := FALSE, SyncCV := 0);
Parameters.Regulation.SupplyAir.Control.SP_HighSpeed := Parameters.Regulation.SupplyAir.Control.SP;
Parameters.Regulation.ExtractAir.Control.SP_HighSpeed := Parameters.Regulation.ExtractAir.Control.SP;
RemoteOrderToSend.SupplySP := Parameters.Regulation.SupplyAir.Control.SP;
RemoteOrderToSend.ExtractSP := Parameters.Regulation.ExtractAir.Control.SP;
END_METHOD

METHOD MasterSlave_DUAL_START_ENTRY : BOOL
VAR_INPUT
END_VAR
StateTime.Restart();
Parameters.IO.DOut.T_QM2 := TRUE;
Parameters.IO.DOut.F_QM1 := TRUE;	
Parameters.Regulation.SupplyAir.ControlMode := FanControlTypes.Const;
Parameters.Regulation.ExtractAir.ControlMode := FanControlTypes.Const;
PidControlSupplyAir(Sync := FALSE, SyncCV := 0.55);
PidControlExtractAir(Sync := FALSE, SyncCV := 0.65);
PidControlSupplyAir(Sync := TRUE, SyncCV := 0.55);
PidControlExtractAir(Sync := TRUE, SyncCV := 0.65);
END_METHOD

METHOD MasterSlave_EVEN_WEEK_DO : BOOL
VAR_INPUT
END_VAR
IF RemoteStatusData.RemoteStatus.State = systemStates.Run THEN
	Parameters.Regulation.SupplyAir.Control.SP := 0;
	Parameters.Regulation.ExtractAir.Control.SP := 0;
	Parameters.Regulation.SupplyAir.Control.SP_HighSpeed := Parameters.Regulation.SupplyAir.Control.SP;
	Parameters.Regulation.ExtractAir.Control.SP_HighSpeed := Parameters.Regulation.ExtractAir.Control.SP;	
END_IF
RemoteOrderToSend.SupplySP := PidControlSupplyAir(Sync := FALSE, SyncCV := 0);
RemoteOrderToSend.ExtractSP := PidControlExtractAir(Sync := FALSE, SyncCV := 0);
END_METHOD

METHOD MasterSlave_EVEN_WEEK_ENTRY : BOOL
VAR_INPUT
END_VAR
//Parameters.IO.DOut.T_QM2 := FALSE;
//Parameters.IO.DOut.F_QM1 := FALSE;
END_METHOD

ACTION MasterSlave_IDLE_ENTRY:
StateTime.Restart();
Tags.Status.MasterActive := TRUE;
END_ACTION

METHOD MasterSlave_IDLE_ENTRY_1 : BOOL
VAR_INPUT
END_VAR
Parameters.Regulation.SupplyAir.ControlMode := FanControlTypes.Const;
Parameters.Regulation.ExtractAir.ControlMode := FanControlTypes.Const;
Parameters.Regulation.SupplyAir.Control.SP := 0;
Parameters.Regulation.ExtractAir.Control.SP := 0;
Parameters.Regulation.SupplyAir.Control.SP_HighSpeed := Parameters.Regulation.SupplyAir.Control.SP;
Parameters.Regulation.ExtractAir.Control.SP_HighSpeed := Parameters.Regulation.ExtractAir.Control.SP;
Tags.Settings.RemoteOrder.SupplySP := 0;
Tags.Settings.RemoteOrder.ExtractSP := 0;
END_METHOD

METHOD MasterSlave_LOCAL_ENTRY : BOOL
VAR_INPUT
END_VAR
Parameters.System.Operation.EN := TRUE;
Parameters.Regulation.SupplyAir.ControlMode := FanControlTypes.Pressure;
Parameters.Regulation.ExtractAir.ControlMode := FanControlTypes.Pressure;
Parameters.Regulation.SupplyAir.Control.SP := GetSetPointSupply();
Parameters.Regulation.ExtractAir.Control.SP := GetSetPointExtract();
Parameters.Regulation.SupplyAir.Control.SP_HighSpeed := Parameters.Regulation.SupplyAir.Control.SP;
Parameters.Regulation.ExtractAir.Control.SP_HighSpeed := Parameters.Regulation.ExtractAir.Control.SP;
END_METHOD

METHOD MasterSlave_LOCAL_SLAVE_DO : BOOL
VAR_INPUT
END_VAR
Parameters.Regulation.SupplyAir.Control.SP := GetSetPointSupply();
Parameters.Regulation.ExtractAir.Control.SP := GetSetPointExtract();
Parameters.Regulation.SupplyAir.Control.SP_HighSpeed := Parameters.Regulation.SupplyAir.Control.SP;
Parameters.Regulation.ExtractAir.Control.SP_HighSpeed := Parameters.Regulation.ExtractAir.Control.SP;
END_METHOD

METHOD MasterSlave_LOCAL_SLAVE_ENTRY : BOOL
VAR_INPUT
END_VAR
Parameters.Regulation.SupplyAir.ControlMode := FanControlTypes.Pressure;
Parameters.Regulation.ExtractAir.ControlMode := FanControlTypes.Pressure;
(*
Parameters.IO.DOut.T_QM2 := TRUE;
Parameters.IO.DOut.F_QM1 := TRUE;	
*)
END_METHOD

METHOD MasterSlave_MANUAL_ENTRY : BOOL
VAR_INPUT
END_VAR
Parameters.Regulation.SupplyAir.ControlMode := FanControlTypes.Pressure;
Parameters.Regulation.ExtractAir.ControlMode := FanControlTypes.Pressure;
Parameters.Regulation.SupplyAir.Control.SP := GetSetPointSupply();
Parameters.Regulation.ExtractAir.Control.SP := GetSetPointExtract();
Parameters.Regulation.SupplyAir.Control.SP_HighSpeed := Parameters.Regulation.SupplyAir.Control.SP;
Parameters.Regulation.ExtractAir.Control.SP_HighSpeed := Parameters.Regulation.ExtractAir.Control.SP;
END_METHOD

METHOD MasterSlave_MASTER_START_ENTRY : BOOL
VAR_INPUT
END_VAR
StateTime.Restart();
PidControlSupplyAir(Sync := FALSE, SyncCV := 0);
PidControlExtractAir(Sync := false, SyncCV := 0);
PidControlSupplyAir(Sync := TRUE, SyncCV := 0);
PidControlExtractAir(Sync := TRUE, SyncCV := 0);
END_METHOD

METHOD MasterSlave_ODD_WEEK_DO : BOOL
VAR_INPUT
END_VAR
Parameters.Regulation.SupplyAir.Control.SP := PidControlSupplyAir(Sync := FALSE, SyncCV := 0);
Parameters.Regulation.ExtractAir.Control.SP := PidControlExtractAir(Sync := FALSE, SyncCV := 0);
Parameters.Regulation.SupplyAir.Control.SP_HighSpeed := Parameters.Regulation.SupplyAir.Control.SP;
Parameters.Regulation.ExtractAir.Control.SP_HighSpeed := Parameters.Regulation.ExtractAir.Control.SP;
IF Parameters.System.Operation.State = SystemStates.Run THEN
	RemoteOrderToSend.SupplySP := 0;
	RemoteOrderToSend.ExtractSP := 0;	
END_IF
END_METHOD

METHOD MasterSlave_ODD_WEEK_ENTRY : BOOL
VAR_INPUT
END_VAR
//Parameters.IO.DOut.T_QM2 := TRUE;
//Parameters.IO.DOut.F_QM1 := TRUE;
END_METHOD

METHOD MasterSlave_SINGLE_START_ENTRY : BOOL
VAR_INPUT
END_VAR
StateTime.Restart();
Parameters.Regulation.SupplyAir.ControlMode := FanControlTypes.Const;
Parameters.Regulation.ExtractAir.ControlMode := FanControlTypes.Const;
PidControlSupplyAir(Sync := FALSE, SyncCV := 0.55);
PidControlExtractAir(Sync := false, SyncCV := 0.65);
PidControlSupplyAir(Sync := TRUE, SyncCV := 0.55);
PidControlExtractAir(Sync := TRUE, SyncCV := 0.65);
END_METHOD

METHOD MasterSlave_SLAVE_DO : BOOL
VAR_INPUT
END_VAR
VAR
	Supply: LREAL;
	Extract: LREAL;
END_VAR
Parameters.Regulation.SupplyAir.Control.SP := Tags.Settings.RemoteOrder.SupplySP;
Parameters.Regulation.ExtractAir.Control.SP := Tags.Settings.RemoteOrder.ExtractSP;	
Parameters.Regulation.SupplyAir.Control.SP_HighSpeed := Parameters.Regulation.SupplyAir.Control.SP;
Parameters.Regulation.ExtractAir.Control.SP_HighSpeed := Parameters.Regulation.ExtractAir.Control.SP;
(*
IF (Tags.Settings.RemoteOrder.SupplySP = 0) AND (Tags.Settings.RemoteOrder.ExtractSP = 0) THEN
	Parameters.IO.DOut.T_QM2 := FALSE;
	Parameters.IO.DOut.F_QM1 := FALSE;	
ELSE
	Parameters.IO.DOut.T_QM2 := TRUE;
	Parameters.IO.DOut.F_QM1 := TRUE;	
END_IF
*)
END_METHOD

METHOD MasterSlave_SLAVE_ENTRY : BOOL
VAR_INPUT
END_VAR
StateTime.Restart();
Parameters.Regulation.SupplyAir.ControlMode := FanControlTypes.Const;
Parameters.Regulation.ExtractAir.ControlMode := FanControlTypes.Const;
END_METHOD

METHOD MasterSlave_SLAVE_IDLE_ENTRY : BOOL
VAR_INPUT
END_VAR
StateTime.Restart();
END_METHOD

METHOD MasterSlave_State1_DO : BOOL
VAR_INPUT
END_VAR
Parameters.Regulation.SupplyAir.Control.SP := GetSetPointSupply();
Parameters.Regulation.ExtractAir.Control.SP := GetSetPointExtract();
Parameters.Regulation.SupplyAir.Control.SP_HighSpeed := Parameters.Regulation.SupplyAir.Control.SP;
Parameters.Regulation.ExtractAir.Control.SP_HighSpeed := Parameters.Regulation.ExtractAir.Control.SP;
END_METHOD

METHOD MasterSlave_State1_ENTRY : BOOL
VAR_INPUT
END_VAR
Parameters.Regulation.SupplyAir.ControlMode := FanControlTypes.Pressure;
Parameters.Regulation.ExtractAir.ControlMode := FanControlTypes.Pressure;
//Parameters.IO.DOut.T_QM2 := TRUE;
//Parameters.IO.DOut.F_QM1 := TRUE;
END_METHOD

METHOD MasterSlave_State1_ENTRY_1 : BOOL
VAR_INPUT
END_VAR
Parameters.Regulation.SupplyAir.Control.SP := GetSetPointSupply();
Parameters.Regulation.ExtractAir.Control.SP := GetSetPointExtract();
Parameters.Regulation.SupplyAir.Control.SP_HighSpeed := Parameters.Regulation.SupplyAir.Control.SP;
Parameters.Regulation.ExtractAir.Control.SP_HighSpeed := Parameters.Regulation.ExtractAir.Control.SP;
END_METHOD

METHOD PidControlExtractAir : LREAL
VAR_INPUT
	Sync: BOOL;
	SyncCV: LREAL := 0;
END_VAR
VAR_INST
	pid: PidController;
	pidOutput: LREAL;
END_VAR
pid(	SP := GetSetPointExtract(), 
		PV := Parameters.IO.AIn.F_BP1, 
		Sync := Sync, 
		SyncCV := SyncCV,
		P := Tags.Settings.Kp, 
		I := Tags.Settings.fTn, 
		DampingTime := Tags.Settings.fTv, 
		CV => pidOutput);
PidControlExtractAir := LimitValue(pidOutput * 100, 0, 100);
END_METHOD

METHOD PidControlSupplyAir : LREAL
VAR_INPUT
	Sync: BOOL;
	SyncCV: LREAL := 0;
END_VAR
VAR_INST
	pid: PidController;
	pidOutput: LREAL;
END_VAR
pid(	SP := GetSetPointSupply(), 
		PV := Parameters.IO.AIn.T_BP1, 
		Sync := Sync, 
		SyncCV := SyncCV,
		P := Tags.Settings.Kp, 
		I := Tags.Settings.fTn, 
		DampingTime := Tags.Settings.fTv, 
		CV => pidOutput);
PidControlSupplyAir := LimitValue(pidOutput * 100, 0, 100);
END_METHOD

METHOD ReadFromRemote : RemoteStatusData
VAR_INPUT
END_VAR
VAR_INST
	ReadAdsSymbol:FB_ReadAdsSymByName;	
	RemoteStatus: ParallelUnitsStatus;
	ValidTOF: TOF;
END_VAR
IF NOT ReadAdsSymbol.bBusy THEN
	ReadAdsSymbol(	bRead		:=	TRUE,
					sNetId		:=	Tags.Settings.RemoteAmsId,
					nPort		:=	851,
					sVarName	:=	'ADS_ParallelUnits.Tags.Status',
					nDestAddr	:=	ADR(RemoteStatus),
					nLen		:=	SIZEOF(RemoteStatus),
					tTimeout	:=	DEFAULT_ADS_TIMEOUT,
					eComMode	:=	eAdsComModeFastCom);
END_IF;
ReadAdsSymbol(bRead := FALSE);
ValidTOF(IN := NOT ReadAdsSymbol.bBusy AND NOT ReadAdsSymbol.bError, PT := T#5S);
ReadFromRemote.Valid := ValidTOF.Q;
ReadFromRemote.RemoteStatus := RemoteStatus;
END_METHOD

METHOD SlaveCanRun : BOOL
VAR_INPUT
END_VAR
SlaveCanRun := RemoteStatusData.RemoteStatus.CanBeRunnable;
END_METHOD

METHOD TransferToRemote : BOOL
VAR_INPUT
	sNetId: T_AmsNetID;
	Src: REFERENCE TO RemoteOrder;
	Dest: string;
END_VAR
VAR_INST
	WriteAdsSymbol: FB_WriteAdsSymByName;	
END_VAR
IF NOT WriteAdsSymbol.bBusy THEN
	WriteAdsSymbol(	bWrite		:=	TRUE,
					sNetId		:=	Tags.Settings.RemoteAmsId,
					nPort		:=	851,
					sVarName	:=	Dest,
					nSrcAddr	:=	ADR(Src),
					nLen		:=	SIZEOF(Src),
					tTimeout	:=	DEFAULT_ADS_TIMEOUT,
					eComMode	:=	eAdsComModeFastCom);
END_IF;
WriteAdsSymbol(bWrite := FALSE);
TransferToRemote := NOT WriteAdsSymbol.bBusy AND NOT WriteAdsSymbol.bError;
END_METHOD

END_FUNCTION_BLOCK

